C01842=1151.994,50.218,-50.534,-179.726,6.301,149.061
C01843=1151.990,50.468,-50.550,-179.724,6.302,149.061
C01844=1151.985,50.717,-50.567,-179.722,6.303,149.060
C01845=1151.979,50.966,-50.582,-179.718,6.304,149.060
C01846=1151.975,51.216,-50.597,-179.716,6.305,149.059
C01847=1151.970,51.465,-50.613,-179.713,6.307,149.059
C01848=1151.964,51.715,-50.629,-179.711,6.307,149.058
C01849=1151.960,51.965,-50.645,-179.708,6.309,149.058
C01850=1151.955,52.214,-50.661,-179.705,6.309,149.057
C01851=1151.950,52.463,-50.676,-179.703,6.310,149.057
C01852=1151.945,52.713,-50.692,-179.700,6.312,149.056
C01853=1151.940,52.962,-50.707,-179.698,6.312,149.056
C01854=1151.934,53.212,-50.723,-179.695,6.314,149.055
C01855=1151.929,53.481,-50.740,-179.692,6.315,149.054
C01856=1151.924,53.749,-50.757,-179.689,6.316,149.054
C01857=1151.918,54.018,-50.774,-179.686,6.318,149.053
C01858=1151.913,54.286,-50.791,-179.683,6.319,149.053
C01859=1151.908,54.535,-50.808,-179.681,6.320,149.052
C01860=1151.904,54.785,-50.823,-179.678,6.321,149.052
C01861=1151.898,55.034,-50.839,-179.676,6.322,149.051
C01862=1151.894,55.284,-50.855,-179.673,6.323,149.051
C01863=1151.888,55.533,-50.871,-179.670,6.324,149.050
C01864=1151.883,55.783,-50.887,-179.668,6.326,149.050
C01865=1151.878,56.032,-50.903,-179.665,6.326,149.049
C01866=1151.873,56.282,-50.919,-179.662,6.328,149.048
C01867=1151.868,56.532,-50.935,-179.660,6.329,149.048
C01868=1151.863,56.780,-50.951,-179.657,6.330,149.047
C01869=1151.858,57.030,-50.967,-179.655,6.331,149.047
C01870=1151.853,57.280,-50.983,-179.651,6.332,149.046
C01871=1151.848,57.529,-50.999,-179.649,6.333,149.046
C01872=1151.843,57.779,-51.015,-179.646,6.335,149.045
C01873=1151.838,58.028,-51.031,-179.644,6.335,149.045
C01874=1151.833,58.277,-51.047,-179.641,6.337,149.044
C01875=1151.828,58.526,-51.063,-179.638,6.337,149.044
C01876=1151.823,58.776,-51.079,-179.636,6.339,149.043
C01877=1151.818,59.025,-51.096,-179.634,6.340,149.043
C01878=1151.813,59.275,-51.111,-179.630,6.341,149.042
C01879=1151.808,59.525,-51.127,-179.628,6.342,149.042
C01880=1151.803,59.774,-51.144,-179.625,6.344,149.041
C01881=1151.798,60.024,-51.159,-179.623,6.344,149.041
C01882=1151.793,60.273,-51.176,-179.620,6.346,149.040
C01883=1151.788,60.523,-51.192,-179.617,6.346,149.039
C01884=1151.783,60.771,-51.208,-179.615,6.348,149.039
C01885=1151.779,61.021,-51.225,-179.613,6.349,149.039
C01886=1151.773,61.270,-51.240,-179.609,6.350,149.038
C01887=1151.769,61.520,-51.257,-179.607,6.351,149.037
C01888=1151.764,61.769,-51.273,-179.604,6.352,149.037
C01889=1151.759,62.019,-51.289,-179.602,6.353,149.036
C01890=1151.754,62.268,-51.305,-179.599,6.355,149.036
C01891=1151.749,62.518,-51.322,-179.596,6.356,149.035
C01892=1151.743,62.767,-51.338,-179.594,6.357,149.035
C01893=1151.739,63.017,-51.354,-179.591,6.358,149.034
C01894=1151.734,63.266,-51.371,-179.588,6.359,149.034
C01895=1151.729,63.516,-51.387,-179.585,6.361,149.033
C01896=1151.724,63.764,-51.403,-179.583,6.361,149.033
C01897=1151.719,64.014,-51.420,-179.580,6.363,149.032
C01898=1151.714,64.263,-51.435,-179.578,6.364,149.032
C01899=1151.709,64.513,-51.452,-179.575,6.365,149.031
C01900=1151.704,64.762,-51.469,-179.573,6.366,149.031
C01901=1151.699,65.012,-51.485,-179.570,6.367,149.030
C01902=1151.694,65.261,-51.501,-179.567,6.369,149.030
C01903=1151.689,65.510,-51.518,-179.564,6.370,149.029
C01904=1151.685,65.760,-51.534,-179.562,6.371,149.029
C01905=1151.679,66.009,-51.551,-179.559,6.372,149.028
C01906=1151.674,66.259,-51.567,-179.556,6.373,149.028
C01907=1151.669,66.508,-51.583,-179.554,6.374,149.027
C01908=1151.665,66.757,-51.600,-179.551,6.376,149.027
C01909=1151.660,67.007,-51.616,-179.548,6.377,149.026
C01910=1151.654,67.256,-51.633,-179.546,6.378,149.025
C01911=1151.649,67.506,-51.650,-179.543,6.379,149.025
C01912=1151.644,67.755,-51.666,-179.541,6.380,149.025
C01913=1151.640,68.004,-51.683,-179.537,6.382,149.024
C01914=1151.634,68.255,-51.699,-179.535,6.382,149.023
C01915=1151.629,68.503,-51.715,-179.533,6.384,149.023
C01916=1151.625,68.753,-51.732,-179.529,6.385,149.022
C01917=1151.620,69.002,-51.748,-179.527,6.386,149.022
C01918=1151.615,69.251,-51.766,-179.524,6.388,149.022
C01919=1151.610,69.501,-51.782,-179.522,6.388,149.021
C01920=1151.605,69.750,-51.799,-179.519,6.390,149.020
C01921=1151.599,70.000,-51.815,-179.516,6.392,149.020
C01922=1151.595,70.250,-51.832,-179.514,6.392,149.019
C01923=1151.590,70.498,-51.848,-179.511,6.394,149.019
C01924=1151.585,70.748,-51.865,-179.509,6.395,149.018
C01925=1151.580,70.998,-51.882,-179.506,6.396,149.018
C01926=1151.575,71.246,-51.898,-179.503,6.398,149.017
C01927=1151.570,71.496,-51.916,-179.501,6.399,149.017
C01928=1151.565,71.746,-51.932,-179.497,6.400,149.016
C01929=1151.560,71.994,-51.949,-179.495,6.401,149.016
C01930=1151.555,72.244,-51.966,-179.493,6.402,149.015
C01931=1151.551,72.494,-51.983,-179.489,6.404,149.015
C01932=1151.546,72.743,-51.999,-179.487,6.405,149.014
C01933=1151.540,72.992,-52.016,-179.484,6.406,149.014
C01934=1151.536,73.242,-52.033,-179.482,6.407,149.013
C01935=1151.530,73.491,-52.050,-179.479,6.408,149.013
C01936=1151.526,73.740,-52.066,-179.476,6.410,149.012
C01937=1151.521,73.990,-52.083,-179.474,6.411,149.012
C01938=1151.516,74.240,-52.100,-179.471,6.412,149.011
C01939=1151.511,74.488,-52.117,-179.468,6.413,149.011
C01940=1151.506,74.738,-52.134,-179.466,6.414,149.010
C01941=1151.501,74.988,-52.151,-179.463,6.416,149.010
C01942=1151.496,75.238,-52.168,-179.461,6.417,149.009
C01943=1151.491,75.486,-52.185,-179.458,6.418,149.009
C01944=1151.487,75.735,-52.202,-179.455,6.420,149.008
C01945=1151.481,75.985,-52.219,-179.453,6.421,149.008
C01946=1151.477,76.234,-52.235,-179.449,6.422,149.007
C01947=1151.471,76.484,-52.252,-179.447,6.424,149.007
C01948=1151.467,76.733,-52.269,-179.445,6.425,149.006
C01949=1151.461,76.983,-52.286,-179.441,6.426,149.006
C01950=1151.457,77.232,-52.304,-179.439,6.427,149.005
C01951=1151.451,77.481,-52.321,-179.436,6.428,149.005
C01952=1151.447,77.730,-52.337,-179.433,6.430,149.004
C01953=1151.442,77.980,-52.355,-179.431,6.431,149.004
C01954=1151.436,78.230,-52.372,-179.428,6.432,149.003
C01955=1151.432,78.479,-52.389,-179.425,6.434,149.003
C01956=1151.426,78.728,-52.406,-179.423,6.435,149.002
C01957=1151.422,78.977,-52.423,-179.420,6.436,149.002
C01958=1151.417,79.227,-52.440,-179.417,6.437,149.001
C01959=1151.412,79.495,-52.459,-179.414,6.439,149.001
C01960=1151.406,79.763,-52.477,-179.412,6.440,149.000
C01961=1151.401,80.032,-52.496,-179.409,6.441,149.000
C01962=1151.396,80.300,-52.514,-179.406,6.443,148.999
C01963=1151.391,80.550,-52.531,-179.403,6.444,148.999
C01964=1151.386,80.799,-52.549,-179.401,6.445,148.998
C01965=1151.381,81.048,-52.566,-179.398,6.447,148.998
C01966=1151.376,81.298,-52.583,-179.395,6.448,148.997
C01967=1151.372,81.547,-52.600,-179.393,6.449,148.997
C01968=1151.367,81.797,-52.617,-179.390,6.451,148.996
C01969=1151.361,82.045,-52.635,-179.387,6.452,148.996
C01970=1151.357,82.295,-52.652,-179.384,6.454,148.995
C01971=1151.351,82.545,-52.669,-179.382,6.455,148.995
C01972=1151.346,82.794,-52.687,-179.379,6.456,148.994
C01973=1151.342,83.043,-52.704,-179.376,6.458,148.994
C01974=1151.337,83.292,-52.722,-179.374,6.458,148.993
C01975=1151.332,83.542,-52.739,-179.371,6.460,148.993
C01976=1151.327,83.792,-52.756,-179.368,6.461,148.992
C01977=1151.322,84.041,-52.774,-179.366,6.462,148.992
C01978=1151.317,84.290,-52.790,-179.363,6.464,148.991
C01979=1151.312,84.539,-52.808,-179.360,6.465,148.991
C01980=1151.307,84.789,-52.825,-179.358,6.466,148.990
C01981=1151.302,85.038,-52.843,-179.355,6.468,148.990
C01982=1151.297,85.288,-52.860,-179.352,6.470,148.989
C01983=1151.293,85.536,-52.878,-179.349,6.471,148.989
C01984=1151.288,85.786,-52.895,-179.347,6.472,148.988
C01985=1151.283,86.035,-52.913,-179.344,6.473,148.988
C01986=1151.278,86.285,-52.930,-179.341,6.475,148.987
C01987=1151.273,86.534,-52.948,-179.339,6.476,148.987
C01988=1151.268,86.783,-52.966,-179.336,6.477,148.986
C01989=1151.263,87.033,-52.983,-179.333,6.479,148.986
C01990=1151.258,87.282,-53.001,-179.331,6.479,148.985
C01991=1151.253,87.532,-53.018,-179.328,6.481,148.985
C01992=1151.249,87.781,-53.035,-179.325,6.483,148.984
C01993=1151.244,88.030,-53.053,-179.322,6.484,148.984
C01994=1151.239,88.280,-53.071,-179.320,6.485,148.983
C01995=1151.233,88.528,-53.088,-179.317,6.487,148.983
C01996=1151.228,88.778,-53.106,-179.314,6.488,148.983
C01997=1151.224,89.027,-53.123,-179.311,6.490,148.982
C01998=1151.219,89.276,-53.141,-179.309,6.491,148.981
C01999=1151.214,89.525,-53.159,-179.306,6.492,148.981
C02000=1151.209,89.775,-53.176,-179.303,6.494,148.981
C02001=1151.204,90.024,-53.194,-179.301,6.494,148.980
C02002=1151.200,90.274,-53.213,-179.298,6.496,148.980
C02003=1151.194,90.524,-53.230,-179.295,6.498,148.979
C02004=1151.190,90.773,-53.248,-179.293,6.499,148.979
C02005=1151.185,91.022,-53.265,-179.290,6.500,148.978
C02006=1151.180,91.271,-53.283,-179.287,6.502,148.978
C02007=1151.175,91.521,-53.300,-179.284,6.503,148.977
C02008=1151.170,91.770,-53.318,-179.282,6.505,148.977
C02009=1151.165,92.019,-53.336,-179.279,6.506,148.976
C02010=1151.160,92.269,-53.354,-179.276,6.507,148.976
C02011=1151.156,92.518,-53.372,-179.274,6.509,148.975
C02012=1151.150,92.768,-53.390,-179.271,6.511,148.975
C02013=1151.145,93.017,-53.408,-179.268,6.511,148.974
C02014=1151.141,93.266,-53.426,-179.266,6.513,148.974
C02015=1151.136,93.515,-53.443,-179.263,6.514,148.973
C02016=1151.131,93.764,-53.461,-179.260,6.516,148.973
C02017=1151.126,94.013,-53.479,-179.257,6.517,148.972
C02018=1151.121,94.263,-53.497,-179.255,6.518,148.972
C02019=1151.116,94.513,-53.515,-179.252,6.520,148.972
C02020=1151.111,94.762,-53.533,-179.249,6.522,148.971
C02021=1151.106,95.011,-53.551,-179.246,6.523,148.970
C02022=1151.102,95.261,-53.569,-179.244,6.524,148.970
C02023=1151.097,95.510,-53.587,-179.241,6.526,148.970
C02024=1151.092,95.759,-53.605,-179.238,6.527,148.969
C02025=1151.087,96.008,-53.623,-179.235,6.529,148.969
C02026=1151.082,96.257,-53.641,-179.233,6.529,148.968
C02027=1151.077,96.506,-53.659,-179.230,6.531,148.968
C02028=1151.073,96.756,-53.677,-179.228,6.533,148.967
C02029=1151.068,97.006,-53.695,-179.224,6.534,148.967
C02030=1151.063,97.255,-53.713,-179.222,6.536,148.966
C02031=1151.058,97.504,-53.731,-179.220,6.537,148.966
C02032=1151.053,97.753,-53.749,-179.217,6.538,148.965
C02033=1151.048,98.002,-53.767,-179.214,6.540,148.965
C02034=1151.043,98.251,-53.785,-179.211,6.541,148.964
C02035=1151.038,98.502,-53.804,-179.208,6.543,148.964
C02036=1151.033,98.751,-53.822,-179.206,6.544,148.964
C02037=1151.028,99.000,-53.840,-179.203,6.546,148.963
C02038=1151.023,99.249,-53.858,-179.200,6.547,148.962
C02039=1151.019,99.498,-53.876,-179.197,6.549,148.962
C02040=1151.014,99.748,-53.895,-179.195,6.550,148.962
C02041=1151.010,99.997,-53.913,-179.192,6.551,148.961
C02042=1151.004,100.246,-53.932,-179.190,6.553,148.961
C02043=1150.999,100.495,-53.950,-179.187,6.554,148.960
C02044=1150.994,100.745,-53.968,-179.184,6.556,148.960
C02045=1150.990,100.994,-53.986,-179.181,6.558,148.959
C02046=1150.985,101.244,-54.004,-179.179,6.559,148.959
C02047=1150.980,101.492,-54.023,-179.176,6.560,148.959
C02048=1150.975,101.742,-54.041,-179.173,6.562,148.958
C02049=1150.970,101.992,-54.060,-179.170,6.563,148.957
C02050=1150.965,102.241,-54.077,-179.168,6.565,148.957
C02051=1150.960,102.490,-54.095,-179.165,6.567,148.957
C02052=1150.955,102.739,-54.115,-179.162,6.567,148.956
C02053=1150.951,102.989,-54.133,-179.159,6.569,148.956
C02054=1150.946,103.238,-54.151,-179.157,6.571,148.955
C02055=1150.941,103.487,-54.169,-179.154,6.572,148.955
C02056=1150.936,103.736,-54.188,-179.151,6.574,148.954
C02057=1150.931,103.986,-54.207,-179.149,6.576,148.954
C02058=1150.926,104.235,-54.225,-179.146,6.576,148.953
C02059=1150.922,104.483,-54.243,-179.143,6.578,148.953
C02060=1150.916,104.733,-54.262,-179.140,6.580,148.952
C02061=1150.912,104.983,-54.280,-179.138,6.581,148.952
C02062=1150.907,105.231,-54.299,-179.135,6.583,148.952
C02063=1150.901,105.500,-54.319,-179.132,6.584,148.951
C02064=1150.896,105.768,-54.338,-179.129,6.586,148.951
C02065=1150.891,106.037,-54.359,-179.126,6.587,148.950
C02066=1150.886,106.305,-54.379,-179.123,6.589,148.950
C02067=1150.881,106.555,-54.397,-179.120,6.591,148.949
C02068=1150.877,106.804,-54.417,-179.118,6.592,148.949
C02069=1150.872,107.053,-54.435,-179.115,6.594,148.948
C02070=1150.866,107.303,-54.453,-179.112,6.595,148.948
C02071=1150.862,107.552,-54.472,-179.110,6.596,148.947
C02072=1150.857,107.801,-54.490,-179.107,6.598,148.947
C02073=1150.852,108.050,-54.509,-179.104,6.600,148.946
C02074=1150.848,108.300,-54.528,-179.101,6.601,148.946
C02075=1150.842,108.549,-54.547,-179.099,6.603,148.946
C02076=1150.837,108.798,-54.565,-179.096,6.604,148.945
C02077=1150.833,109.047,-54.584,-179.093,6.606,148.945
C02078=1150.828,109.296,-54.603,-179.091,6.607,148.944
C02079=1150.823,109.545,-54.621,-179.088,6.609,148.944
C02080=1150.818,109.795,-54.640,-179.085,6.610,148.943
C02081=1150.813,110.044,-54.659,-179.083,6.612,148.943
C02082=1150.808,110.294,-54.678,-179.079,6.613,148.942
C02083=1150.804,110.543,-54.697,-179.077,6.615,148.942
C02084=1150.798,110.791,-54.716,-179.074,6.617,148.942
C02085=1150.794,111.041,-54.734,-179.071,6.618,148.941
C02086=1150.789,111.290,-54.754,-179.069,6.619,148.941
C02087=1150.784,111.540,-54.772,-179.066,6.621,148.940
C02088=1150.779,111.789,-54.791,-179.063,6.622,148.940
C02089=1150.775,112.037,-54.810,-179.060,6.624,148.939
C02090=1150.769,112.288,-54.829,-179.058,6.626,148.939
C02091=1150.765,112.536,-54.848,-179.055,6.627,148.938
C02092=1150.760,112.786,-54.867,-179.052,6.629,148.938
C02093=1150.755,113.035,-54.885,-179.049,6.631,148.938
C02094=1150.750,113.285,-54.905,-179.047,6.633,148.937
C02095=1150.746,113.533,-54.924,-179.044,6.634,148.937
C02096=1150.741,113.783,-54.942,-179.041,6.635,148.936
C02097=1150.736,114.032,-54.961,-179.039,6.636,148.936
C02098=1150.731,114.281,-54.981,-179.036,6.638,148.935
C02099=1150.726,114.530,-55.000,-179.033,6.640,148.935
C02100=1150.721,114.779,-55.018,-179.031,6.642,148.935
C02101=1150.716,115.029,-55.038,-179.028,6.643,148.934
C02102=1150.712,115.278,-55.056,-179.025,6.645,148.934
C02103=1150.707,115.527,-55.076,-179.022,6.646,148.933
C02104=1150.701,115.777,-55.095,-179.019,6.648,148.933
C02105=1150.697,116.026,-55.114,-179.016,6.650,148.932
C02106=1150.692,116.275,-55.133,-179.014,6.651,148.932
C02107=1150.688,116.524,-55.152,-179.011,6.653,148.931
C02108=1150.683,116.773,-55.171,-179.008,6.655,148.931
C02109=1150.678,117.022,-55.191,-179.006,6.656,148.931
C02110=1150.673,117.272,-55.209,-179.003,6.657,148.930
C02111=1150.668,117.521,-55.229,-179.000,6.659,148.930
C02112=1150.664,117.771,-55.248,-178.997,6.660,148.929
C02113=1150.659,118.019,-55.267,-178.995,6.662,148.929
C02114=1150.654,118.269,-55.287,-178.992,6.664,148.928
C02115=1150.649,118.518,-55.306,-178.989,6.666,148.928
C02116=1150.644,118.767,-55.326,-178.987,6.667,148.928
C02117=1150.640,119.016,-55.344,-178.984,6.669,148.927
C02118=1150.635,119.265,-55.364,-178.981,6.671,148.927
C02119=1150.629,119.514,-55.383,-178.978,6.672,148.926
C02120=1150.625,119.764,-55.402,-178.975,6.674,148.926
C02121=1150.621,120.013,-55.422,-178.973,6.675,148.925
C02122=1150.615,120.262,-55.441,-178.970,6.677,148.925
C02123=1150.611,120.512,-55.461,-178.967,6.679,148.925
C02124=1150.605,120.760,-55.480,-178.964,6.681,148.924
C02125=1150.601,121.010,-55.499,-178.962,6.682,148.924
C02126=1150.597,121.259,-55.519,-178.959,6.684,148.923
C02127=1150.591,121.508,-55.538,-178.956,6.686,148.923
C02128=1150.586,121.758,-55.558,-178.953,6.687,148.923
C02129=1150.582,122.006,-55.577,-178.950,6.689,148.922
C02130=1150.577,122.256,-55.596,-178.948,6.690,148.922
C02131=1150.572,122.505,-55.616,-178.945,6.691,148.921
C02132=1150.567,122.754,-55.635,-178.943,6.693,148.921
C02133=1150.562,123.004,-55.655,-178.940,6.695,148.920
C02134=1150.558,123.253,-55.674,-178.937,6.696,148.920
C02135=1150.553,123.501,-55.694,-178.935,6.698,148.920
C02136=1150.549,123.751,-55.714,-178.932,6.700,148.919
C02137=1150.544,124.000,-55.733,-178.929,6.701,148.919
C02138=1150.538,124.249,-55.753,-178.926,6.703,148.918
C02139=1150.534,124.499,-55.772,-178.924,6.705,148.918
C02140=1150.529,124.748,-55.792,-178.921,6.707,148.918
C02141=1150.524,124.997,-55.812,-178.918,6.708,148.917
C02142=1150.519,125.246,-55.831,-178.915,6.710,148.917
C02143=1150.515,125.496,-55.851,-178.912,6.711,148.916
C02144=1150.510,125.744,-55.870,-178.910,6.713,148.916
C02145=1150.505,125.993,-55.890,-178.907,6.715,148.915
C02146=1150.501,126.243,-55.910,-178.904,6.716,148.915
C02147=1150.495,126.492,-55.929,-178.901,6.718,148.915
C02148=1150.491,126.741,-55.949,-178.899,6.720,148.914
C02149=1150.486,126.990,-55.969,-178.896,6.722,148.914
C02150=1150.481,127.240,-55.989,-178.893,6.723,148.913
C02151=1150.476,127.489,-56.008,-178.891,6.725,148.913
C02152=1150.472,127.738,-56.028,-178.888,6.727,148.913
C02153=1150.467,127.987,-56.048,-178.885,6.728,148.912
C02154=1150.462,128.237,-56.068,-178.882,6.730,148.912
C02155=1150.457,128.485,-56.088,-178.880,6.732,148.911
C02156=1150.452,128.735,-56.107,-178.877,6.734,148.911
C02157=1150.448,128.984,-56.127,-178.874,6.735,148.911
C02158=1150.443,129.233,-56.148,-178.871,6.737,148.910
C02159=1150.438,129.482,-56.167,-178.868,6.738,148.910
C02160=1150.433,129.731,-56.187,-178.865,6.741,148.909
C02161=1150.429,129.981,-56.207,-178.862,6.743,148.909
C02162=1150.424,130.230,-56.226,-178.860,6.744,148.908
C02163=1150.419,130.478,-56.246,-178.857,6.746,148.908
C02164=1150.414,130.728,-56.266,-178.854,6.748,148.908
C02165=1150.410,130.977,-56.287,-178.851,6.749,148.907
C02166=1150.405,131.226,-56.306,-178.849,6.751,148.907
C02167=1150.400,131.495,-56.329,-178.846,6.753,148.906
C02168=1150.395,131.763,-56.350,-178.843,6.755,148.906
C02169=1150.389,132.032,-56.371,-178.840,6.757,148.906
C02170=1150.384,132.300,-56.393,-178.837,6.758,148.905
C02171=1150.380,132.550,-56.413,-178.834,6.760,148.905
C02172=1150.375,132.798,-56.433,-178.831,6.762,148.904
C02173=1150.369,133.048,-56.453,-178.829,6.764,148.904
C02174=1150.365,133.297,-56.473,-178.826,6.765,148.903
C02175=1150.360,133.547,-56.493,-178.823,6.767,148.903
C02176=1150.355,133.796,-56.513,-178.821,6.769,148.903
C02177=1150.351,134.045,-56.534,-178.818,6.770,148.902
C02178=1150.346,134.293,-56.553,-178.815,6.772,148.902
C02179=1150.341,134.543,-56.574,-178.812,6.774,148.901
C02180=1150.336,134.792,-56.594,-178.810,6.776,148.901
C02181=1150.331,135.041,-56.614,-178.806,6.778,148.901
C02182=1150.327,135.290,-56.634,-178.804,6.780,148.900
C02183=1150.322,135.539,-56.655,-178.801,6.781,148.900
C02184=1150.317,135.789,-56.675,-178.798,6.783,148.900
C02185=1150.313,136.038,-56.695,-178.796,6.785,148.899
C02186=1150.308,136.286,-56.715,-178.793,6.787,148.899
C02187=1150.303,136.536,-56.735,-178.790,6.788,148.898
C02188=1150.298,136.785,-56.756,-178.787,6.790,148.898
C02189=1150.293,137.034,-56.776,-178.785,6.792,148.898
C02190=1150.289,137.283,-56.797,-178.782,6.793,148.897
C02191=1150.284,137.532,-56.816,-178.779,6.795,148.897
C02192=1150.279,137.782,-56.837,-178.777,6.797,148.896
C02193=1150.274,138.031,-56.858,-178.774,6.799,148.896
C02194=1150.270,138.280,-56.878,-178.771,6.801,148.896
C02195=1150.266,138.529,-56.899,-178.768,6.803,148.895
C02196=1150.260,138.778,-56.919,-178.765,6.805,148.895
C02197=1150.256,139.027,-56.939,-178.762,6.806,148.894
C02198=1150.251,139.276,-56.960,-178.760,6.808,148.894
C02199=1150.246,139.526,-56.981,-178.757,6.810,148.894
C02200=1150.242,139.775,-57.001,-178.754,6.811,148.893
C02201=1150.237,140.023,-57.021,-178.752,6.813,148.893
C02202=1150.232,140.273,-57.042,-178.749,6.815,148.893
C02203=1150.227,140.522,-57.062,-178.746,6.817,148.892
C02204=1150.222,140.772,-57.083,-178.743,6.819,148.892
C02205=1150.218,141.021,-57.103,-178.740,6.821,148.891
C02206=1150.213,141.269,-57.124,-178.738,6.823,148.891
C02207=1150.208,141.519,-57.145,-178.735,6.825,148.891
C02208=1150.204,141.768,-57.165,-178.732,6.826,148.890
C02209=1150.198,142.017,-57.186,-178.730,6.828,148.890
C02210=1150.194,142.266,-57.206,-178.727,6.830,148.890
C02211=1150.189,142.515,-57.227,-178.724,6.831,148.889
C02212=1150.184,142.764,-57.248,-178.721,6.834,148.889
C02213=1150.180,143.013,-57.268,-178.718,6.836,148.889
C02214=1150.175,143.262,-57.289,-178.716,6.837,148.888
C02215=1150.170,143.511,-57.309,-178.713,6.839,148.888
C02216=1150.165,143.760,-57.330,-178.710,6.841,148.887
C02217=1150.161,144.009,-57.351,-178.707,6.843,148.887
C02218=1150.155,144.259,-57.372,-178.705,6.844,148.887
C02219=1150.151,144.508,-57.392,-178.701,6.847,148.886
C02220=1150.147,144.757,-57.412,-178.699,6.849,148.886
C02221=1150.142,145.005,-57.434,-178.696,6.850,148.885
C02222=1150.137,145.254,-57.455,-178.693,6.852,148.885
C02223=1150.132,145.503,-57.475,-178.691,6.854,148.885
C02224=1150.127,145.753,-57.496,-178.688,6.855,148.884
C02225=1150.122,146.002,-57.517,-178.685,6.857,148.884
C02226=1150.118,146.252,-57.538,-178.682,6.860,148.884
C02227=1150.113,146.501,-57.558,-178.680,6.862,148.883
C02228=1150.109,146.749,-57.580,-178.677,6.863,148.883
C02229=1150.104,146.998,-57.601,-178.674,6.865,148.883
C02230=1150.099,147.247,-57.621,-178.672,6.867,148.882
C02231=1150.095,147.496,-57.642,-178.669,6.869,148.882
C02232=1150.090,147.745,-57.664,-178.666,6.871,148.881
C02233=1150.085,147.994,-57.685,-178.663,6.873,148.881
C02234=1150.081,148.244,-57.705,-178.660,6.875,148.881
C02235=1150.076,148.493,-57.726,-178.657,6.876,148.880
C02236=1150.071,148.742,-57.748,-178.655,6.878,148.880
C02237=1150.066,148.991,-57.768,-178.652,6.880,148.880
C02238=1150.061,149.240,-57.789,-178.649,6.883,148.879
C02239=1150.057,149.489,-57.810,-178.647,6.884,148.879
C02240=1150.052,149.738,-57.831,-178.644,6.886,148.879
C02241=1150.047,149.988,-57.853,-178.641,6.888,148.878
C02242=1150.043,150.237,-57.873,-178.638,6.890,148.878
C02243=1150.038,150.485,-57.895,-178.636,6.891,148.877
C02244=1150.033,150.734,-57.916,-178.632,6.894,148.877
C02245=1150.028,150.983,-57.937,-178.630,6.896,148.877
C02246=1150.023,151.232,-57.958,-178.627,6.897,148.876
C02247=1150.019,151.482,-57.979,-178.624,6.899,148.876
C02248=1150.014,151.731,-58.001,-178.622,6.901,148.876
C02249=1150.009,151.980,-58.021,-178.619,6.904,148.875
C02250=1150.005,152.228,-58.043,-178.616,6.905,148.875
C02251=1150.000,152.478,-58.064,-178.613,6.907,148.875
C02252=1149.995,152.727,-58.086,-178.611,6.909,148.874
C02253=1149.991,152.976,-58.106,-178.608,6.910,148.874
C02254=1149.986,153.225,-58.127,-178.605,6.913,148.874
C02255=1149.981,153.474,-58.149,-178.602,6.915,148.873
C02256=1149.976,153.724,-58.170,-178.599,6.916,148.873
C02257=1149.971,153.972,-58.192,-178.597,6.919,148.873
C02258=1149.967,154.221,-58.213,-178.594,6.920,148.872
C02259=1149.962,154.470,-58.234,-178.591,6.923,148.872
C02260=1149.958,154.719,-58.256,-178.588,6.925,148.872
C02261=1149.952,154.968,-58.277,-178.586,6.926,148.871
C02262=1149.948,155.217,-58.299,-178.583,6.928,148.871
C02263=1149.944,155.467,-58.319,-178.580,6.930,148.870
C02264=1149.939,155.715,-58.341,-178.577,6.933,148.870
C02265=1149.934,155.964,-58.363,-178.575,6.934,148.870
C02266=1149.929,156.213,-58.384,-178.572,6.936,148.869
C02267=1149.925,156.463,-58.406,-178.569,6.938,148.869
C02268=1149.920,156.711,-58.427,-178.566,6.940,148.869
C02269=1149.915,156.961,-58.448,-178.563,6.942,148.868
C02270=1149.911,157.210,-58.470,-178.561,6.944,148.868
C02271=1149.906,157.479,-58.493,-178.557,6.946,148.868
C02272=1149.900,157.747,-58.516,-178.555,6.948,148.867
C02273=1149.895,158.016,-58.540,-178.551,6.951,148.867
C02274=1149.890,158.285,-58.563,-178.549,6.952,148.866
C02275=1149.886,158.534,-58.584,-178.546,6.954,148.866
C02276=1149.881,158.783,-58.606,-178.543,6.957,148.866
C02277=1149.876,159.032,-58.627,-178.540,6.959,148.866
C02278=1149.872,159.282,-58.649,-178.538,6.960,148.865
C02279=1149.867,159.530,-58.671,-178.535,6.962,148.865
C02280=1149.863,159.780,-58.693,-178.532,6.965,148.864
C02281=1149.857,160.029,-58.714,-178.529,6.967,148.864
C02282=1149.853,160.277,-58.736,-178.527,6.968,148.864
C02283=1149.848,160.527,-58.758,-178.524,6.970,148.864
C02284=1149.843,160.775,-58.779,-178.521,6.973,148.863
C02285=1149.839,161.024,-58.801,-178.518,6.974,148.863
C02286=1149.834,161.273,-58.823,-178.515,6.976,148.862
C02287=1149.829,161.522,-58.845,-178.513,6.979,148.862
C02288=1149.825,161.772,-58.866,-178.510,6.981,148.862
C02289=1149.820,162.021,-58.888,-178.507,6.983,148.862
C02290=1149.816,162.270,-58.910,-178.504,6.984,148.861
C02291=1149.811,162.519,-58.931,-178.501,6.987,148.861
C02292=1149.806,162.767,-58.953,-178.499,6.989,148.861
C02293=1149.802,163.017,-58.975,-178.496,6.991,148.860
C02294=1149.796,163.266,-58.997,-178.493,6.993,148.860
C02295=1149.792,163.515,-59.019,-178.490,6.995,148.860
C02296=1149.787,163.764,-59.041,-178.488,6.997,148.859
C02297=1149.783,164.013,-59.063,-178.485,6.999,148.859
C02298=1149.778,164.262,-59.085,-178.482,7.001,148.859
C02299=1149.774,164.511,-59.107,-178.479,7.003,148.858
C02300=1149.769,164.760,-59.129,-178.477,7.005,148.858
C02301=1149.764,165.009,-59.151,-178.473,7.007,148.858
C02302=1149.760,165.258,-59.172,-178.471,7.009,148.857
C02303=1149.754,165.506,-59.195,-178.468,7.011,148.857
C02304=1149.750,165.756,-59.217,-178.466,7.013,148.857
C02305=1149.745,166.004,-59.238,-178.462,7.015,148.856
C02306=1149.740,166.254,-59.260,-178.460,7.017,148.856
C02307=1149.736,166.502,-59.283,-178.457,7.019,148.856
C02308=1149.732,166.751,-59.305,-178.454,7.022,148.855
C02309=1149.726,167.000,-59.327,-178.451,7.023,148.855
C02310=1149.722,167.249,-59.349,-178.449,7.025,148.855
C02311=1149.718,167.499,-59.371,-178.446,7.028,148.855
C02312=1149.713,167.747,-59.393,-178.443,7.030,148.854
C02313=1149.708,167.997,-59.416,-178.441,7.032,148.854
C02314=1149.703,168.245,-59.438,-178.437,7.034,148.854
C02315=1149.699,168.494,-59.460,-178.435,7.036,148.853
C02316=1149.694,168.743,-59.482,-178.432,7.038,148.853
C02317=1149.689,168.993,-59.504,-178.429,7.040,148.853
C02318=1149.684,169.241,-59.527,-178.426,7.042,148.852
C02319=1149.680,169.490,-59.549,-178.424,7.044,148.852
C02320=1149.675,169.739,-59.570,-178.421,7.047,148.852
C02321=1149.670,169.988,-59.593,-178.418,7.049,148.851
C02322=1149.666,170.237,-59.616,-178.415,7.050,148.851
C02323=1149.661,170.486,-59.638,-178.413,7.053,148.851
C02324=1149.656,170.735,-59.660,-178.410,7.055,148.851
C02325=1149.652,170.983,-59.683,-178.407,7.057,148.850
C02326=1149.648,171.233,-59.705,-178.404,7.059,148.850
C02327=1149.643,171.482,-59.727,-178.402,7.061,148.850
C02328=1149.638,171.730,-59.750,-178.399,7.063,148.849
C02329=1149.634,171.980,-59.772,-178.396,7.066,148.849
C02330=1149.628,172.229,-59.794,-178.393,7.067,148.849
C02331=1149.624,172.477,-59.817,-178.391,7.069,148.848
C02332=1149.619,172.727,-59.839,-178.388,7.072,148.848
C02333=1149.615,172.975,-59.862,-178.385,7.074,148.848
C02334=1149.610,173.224,-59.884,-178.383,7.076,148.848
C02335=1149.606,173.474,-59.907,-178.379,7.078,148.847
C02336=1149.601,173.722,-59.929,-178.377,7.080,148.847
C02337=1149.596,173.972,-59.952,-178.373,7.083,148.846
C02338=1149.592,174.221,-59.974,-178.371,7.085,148.846
C02339=1149.586,174.469,-59.997,-178.369,7.086,148.846
C02340=1149.582,174.718,-60.019,-178.365,7.089,148.846
C02341=1149.578,174.968,-60.041,-178.363,7.091,148.845
C02342=1149.573,175.216,-60.064,-178.360,7.093,148.845
C02343=1149.569,175.465,-60.087,-178.357,7.095,148.845
C02344=1149.564,175.714,-60.110,-178.354,7.097,148.844
C02345=1149.559,175.962,-60.132,-178.352,7.100,148.844
C02346=1149.554,176.212,-60.155,-178.349,7.102,148.844
C02347=1149.550,176.461,-60.178,-178.346,7.103,148.844
C02348=1149.545,176.710,-60.200,-178.343,7.106,148.843
C02349=1149.541,176.958,-60.223,-178.341,7.108,148.843
C02350=1149.536,177.207,-60.246,-178.338,7.110,148.843
C02351=1149.532,177.457,-60.268,-178.335,7.113,148.843
C02352=1149.526,177.705,-60.291,-178.332,7.114,148.842
C02353=1149.522,177.954,-60.314,-178.329,7.117,148.842
C02354=1149.517,178.203,-60.336,-178.327,7.119,148.842
C02355=1149.513,178.452,-60.360,-178.324,7.121,148.841
C02356=1149.508,178.700,-60.382,-178.321,7.123,148.841
C02357=1149.503,178.950,-60.405,-178.319,7.125,148.841
C02358=1149.499,179.199,-60.428,-178.315,7.128,148.841
C02359=1149.494,179.448,-60.451,-178.313,7.130,148.840
C02360=1149.489,179.696,-60.474,-178.311,7.132,148.840
C02361=1149.485,179.946,-60.496,-178.307,7.134,148.840
C02362=1149.480,180.195,-60.519,-178.305,7.136,148.839
C02363=1149.476,180.443,-60.542,-178.302,7.139,148.839
C02364=1149.471,180.692,-60.565,-178.299,7.141,148.839
C02365=1149.466,180.941,-60.588,-178.296,7.143,148.838
C02366=1149.462,181.190,-60.611,-178.294,7.145,148.838
C02367=1149.457,181.439,-60.634,-178.291,7.147,148.838
C02368=1149.453,181.688,-60.657,-178.288,7.150,148.838
C02369=1149.449,181.937,-60.680,-178.285,7.152,148.837
C02370=1149.444,182.186,-60.703,-178.282,7.154,148.837
C02371=1149.439,182.434,-60.726,-178.279,7.156,148.837
C02372=1149.435,182.683,-60.749,-178.277,7.159,148.837
C02373=1149.430,182.933,-60.772,-178.274,7.161,148.836
C02374=1149.425,183.182,-60.795,-178.271,7.162,148.836
C02375=1149.420,183.451,-60.821,-178.268,7.165,148.836
C02376=1149.415,183.720,-60.845,-178.265,7.168,148.835
C02377=1149.410,183.990,-60.870,-178.262,7.171,148.835
C02378=1149.405,184.260,-60.895,-178.259,7.172,148.835
C02379=1149.400,184.509,-60.919,-178.256,7.175,148.835
C02380=1149.396,184.757,-60.941,-178.254,7.177,148.834
C02381=1149.391,185.006,-60.965,-178.250,7.179,148.834
C02382=1149.387,185.255,-60.988,-178.248,7.182,148.834
C02383=1149.382,185.505,-61.012,-178.245,7.184,148.833
C02384=1149.378,185.753,-61.034,-178.243,7.186,148.833
C02385=1149.373,186.002,-61.058,-178.239,7.189,148.833
C02386=1149.369,186.251,-61.081,-178.237,7.190,148.833
C02387=1149.363,186.500,-61.104,-178.235,7.193,148.833
C02388=1149.359,186.748,-61.128,-178.231,7.195,148.832
C02389=1149.354,186.997,-61.151,-178.229,7.197,148.832
C02390=1149.349,187.246,-61.175,-178.226,7.200,148.832
C02391=1149.345,187.495,-61.198,-178.223,7.202,148.831
C02392=1149.341,187.744,-61.221,-178.220,7.204,148.831
C02393=1149.336,187.993,-61.244,-178.218,7.206,148.831
C02394=1149.331,188.242,-61.268,-178.215,7.209,148.831
C02395=1149.327,188.490,-61.292,-178.212,7.211,148.830
C02396=1149.322,188.739,-61.315,-178.209,7.213,148.830
C02397=1149.318,188.988,-61.338,-178.207,7.215,148.830
C02398=1149.313,189.237,-61.362,-178.203,7.218,148.830
C02399=1149.308,189.486,-61.385,-178.201,7.220,148.829
C02400=1149.304,189.735,-61.409,-178.198,7.223,148.829
C02401=1149.299,189.984,-61.433,-178.196,7.225,148.829
C02402=1149.294,190.233,-61.456,-178.192,7.227,148.829
C02403=1149.290,190.482,-61.479,-178.190,7.229,148.828
C02404=1149.286,190.730,-61.503,-178.187,7.232,148.828
C02405=1149.281,190.979,-61.526,-178.184,7.234,148.828
C02406=1149.277,191.228,-61.550,-178.181,7.237,148.828
C02407=1149.272,191.477,-61.574,-178.179,7.238,148.827
C02408=1149.268,191.726,-61.597,-178.176,7.241,148.827
C02409=1149.263,191.975,-61.620,-178.173,7.243,148.827
C02410=1149.258,192.223,-61.645,-178.170,7.246,148.827
C02411=1149.253,192.472,-61.668,-178.168,7.248,148.826
C02412=1149.248,192.721,-61.692,-178.164,7.250,148.826
C02413=1149.244,192.970,-61.716,-178.162,7.252,148.826
C02414=1149.239,193.219,-61.739,-178.159,7.255,148.826
C02415=1149.235,193.467,-61.763,-178.157,7.257,148.825
C02416=1149.230,193.716,-61.787,-178.153,7.260,148.825
C02417=1149.226,193.965,-61.811,-178.151,7.262,148.825
C02418=1149.221,194.214,-61.834,-178.148,7.264,148.825
C02419=1149.217,194.462,-61.858,-178.146,7.266,148.825
C02420=1149.212,194.711,-61.881,-178.142,7.269,148.824
C02421=1149.208,194.960,-61.906,-178.140,7.271,148.824
C02422=1149.203,195.209,-61.929,-178.137,7.274,148.824
C02423=1149.198,195.458,-61.954,-178.135,7.276,148.824
C02424=1149.194,195.707,-61.977,-178.131,7.278,148.823
C02425=1149.189,195.956,-62.001,-178.128,7.281,148.823
C02426=1149.185,196.205,-62.025,-178.126,7.283,148.823
C02427=1149.180,196.453,-62.049,-178.123,7.285,148.822
C02428=1149.175,196.702,-62.072,-178.120,7.288,148.822
C02429=1149.171,196.951,-62.097,-178.117,7.290,148.822
C02430=1149.166,197.200,-62.121,-178.115,7.292,148.822
C02431=1149.162,197.449,-62.145,-178.112,7.295,148.822
C02432=1149.157,197.697,-62.169,-178.110,7.297,148.821
C02433=1149.153,197.946,-62.193,-178.106,7.299,148.821
C02434=1149.148,198.195,-62.217,-178.104,7.302,148.821
C02435=1149.143,198.443,-62.241,-178.101,7.304,148.821
C02436=1149.139,198.693,-62.265,-178.098,7.307,148.821
C02437=1149.135,198.942,-62.289,-178.095,7.309,148.820
C02438=1149.130,199.190,-62.313,-178.092,7.312,148.820
C02439=1149.125,199.439,-62.337,-178.090,7.313,148.820
C02440=1149.120,199.688,-62.361,-178.087,7.316,148.820
C02441=1149.117,199.937,-62.385,-178.084,7.318,148.819
C02442=1149.112,200.186,-62.410,-178.082,7.321,148.819
C02443=1149.107,200.434,-62.434,-178.079,7.323,148.819
C02444=1149.103,200.682,-62.458,-178.076,7.326,148.819
C02445=1149.098,200.931,-62.481,-178.073,7.329,148.819
C02446=1149.094,201.181,-62.506,-178.071,7.330,148.818
C02447=1149.089,201.429,-62.530,-178.068,7.333,148.818
C02448=1149.085,201.678,-62.554,-178.065,7.335,148.818
C02449=1149.080,201.926,-62.579,-178.062,7.338,148.818
C02450=1149.076,202.176,-62.604,-178.059,7.340,148.817
C02451=1149.071,202.425,-62.627,-178.057,7.343,148.817
C02452=1149.066,202.673,-62.652,-178.054,7.345,148.817
C02453=1149.062,202.922,-62.676,-178.051,7.347,148.817
C02454=1149.057,203.171,-62.701,-178.048,7.350,148.816
C02455=1149.053,203.420,-62.725,-178.046,7.352,148.816
C02456=1149.048,203.668,-62.749,-178.043,7.355,148.816
C02457=1149.044,203.917,-62.774,-178.040,7.357,148.816
C02458=1149.039,204.166,-62.798,-178.038,7.359,148.816
C02459=1149.034,204.415,-62.823,-178.034,7.362,148.815
C02460=1149.030,204.663,-62.847,-178.032,7.364,148.815
C02461=1149.026,204.912,-62.871,-178.029,7.367,148.815
C02462=1149.021,205.161,-62.896,-178.026,7.370,148.815
C02463=1149.016,205.409,-62.920,-178.023,7.371,148.815
C02464=1149.012,205.659,-62.945,-178.021,7.374,148.814
C02465=1149.008,205.907,-62.969,-178.018,7.377,148.814
C02466=1149.002,206.156,-62.994,-178.015,7.379,148.814
C02467=1148.999,206.405,-63.018,-178.012,7.382,148.814
C02468=1148.994,206.654,-63.043,-178.010,7.384,148.814
C02469=1148.989,206.902,-63.067,-178.007,7.387,148.813
C02470=1148.985,207.151,-63.092,-178.004,7.389,148.813
C02471=1148.980,207.399,-63.117,-178.001,7.391,148.813
C02472=1148.975,207.648,-63.141,-177.998,7.394,148.813
C02473=1148.971,207.897,-63.166,-177.995,7.397,148.813
C02474=1148.966,208.146,-63.190,-177.993,7.399,148.812
C02475=1148.961,208.394,-63.215,-177.990,7.402,148.812
C02476=1148.958,208.644,-63.240,-177.988,7.403,148.812
C02477=1148.953,208.892,-63.265,-177.985,7.406,148.812
C02478=1148.949,209.141,-63.289,-177.981,7.409,148.812
C02479=1148.943,209.411,-63.317,-177.979,7.412,148.811
C02480=1148.938,209.682,-63.344,-177.975,7.414,148.811
C02481=1148.933,209.952,-63.371,-177.973,7.417,148.811
C02482=1148.929,210.223,-63.398,-177.969,7.420,148.811
C02483=1148.924,210.472,-63.422,-177.967,7.422,148.811
C02484=1148.919,210.720,-63.446,-177.964,7.425,148.811
C02485=1148.915,210.969,-63.472,-177.961,7.428,148.810
C02486=1148.911,211.218,-63.496,-177.959,7.430,148.810
C02487=1148.906,211.467,-63.521,-177.956,7.432,148.810
C02488=1148.901,211.715,-63.547,-177.953,7.434,148.810
C02489=1148.897,211.964,-63.571,-177.951,7.437,148.810
C02490=1148.892,212.213,-63.596,-177.947,7.440,148.809
C02491=1148.888,212.462,-63.621,-177.945,7.442,148.809
C02492=1148.883,212.710,-63.646,-177.942,7.445,148.809
C02493=1148.879,212.958,-63.671,-177.939,7.447,148.809
C02494=1148.874,213.208,-63.696,-177.937,7.449,148.809
C02495=1148.869,213.456,-63.721,-177.934,7.452,148.808
C02496=1148.866,213.705,-63.746,-177.931,7.455,148.808
C02497=1148.861,213.954,-63.770,-177.929,7.457,148.808
C02498=1148.856,214.202,-63.796,-177.926,7.460,148.808
C02499=1148.851,214.451,-63.821,-177.923,7.463,148.808
C02500=1148.848,214.700,-63.846,-177.920,7.465,148.807
C02501=1148.843,214.948,-63.871,-177.918,7.468,148.807
C02502=1148.838,215.197,-63.896,-177.914,7.470,148.807
C02503=1148.833,215.446,-63.921,-177.911,7.473,148.807
C02504=1148.829,215.695,-63.947,-177.909,7.475,148.807
C02505=1148.826,215.943,-63.972,-177.906,7.478,148.807
C02506=1148.820,216.192,-63.997,-177.903,7.481,148.806
C02507=1148.816,216.441,-64.022,-177.901,7.483,148.806
C02508=1148.811,216.689,-64.047,-177.898,7.485,148.806
C02509=1148.807,216.938,-64.073,-177.895,7.488,148.806
C02510=1148.802,217.186,-64.098,-177.893,7.490,148.806
C02511=1148.797,217.436,-64.123,-177.889,7.493,148.805
C02512=1148.793,217.684,-64.148,-177.887,7.496,148.805
C02513=1148.789,217.932,-64.174,-177.884,7.499,148.805
C02514=1148.785,218.182,-64.199,-177.881,7.501,148.805
C02515=1148.780,218.430,-64.224,-177.878,7.503,148.805
C02516=1148.776,218.679,-64.250,-177.876,7.506,148.805
C02517=1148.770,218.927,-64.275,-177.873,7.508,148.805
C02518=1148.766,219.176,-64.300,-177.870,7.511,148.804
C02519=1148.762,219.425,-64.326,-177.867,7.514,148.804
C02520=1148.757,219.673,-64.352,-177.865,7.517,148.804
C02521=1148.753,219.923,-64.377,-177.862,7.519,148.804
C02522=1148.748,220.171,-64.402,-177.859,7.522,148.804
C02523=1148.744,220.419,-64.428,-177.856,7.524,148.804
C02524=1148.740,220.668,-64.453,-177.853,7.527,148.803
C02525=1148.735,220.916,-64.478,-177.851,7.529,148.803
C02526=1148.731,221.165,-64.503,-177.848,7.532,148.803
C02527=1148.727,221.414,-64.529,-177.845,7.535,148.803
C02528=1148.721,221.663,-64.555,-177.843,7.537,148.803
C02529=1148.717,221.912,-64.581,-177.840,7.540,148.803
C02530=1148.713,222.160,-64.607,-177.837,7.543,148.802
C02531=1148.708,222.408,-64.632,-177.834,7.546,148.802
C02532=1148.703,222.657,-64.658,-177.832,7.547,148.802
C02533=1148.699,222.906,-64.683,-177.829,7.550,148.802
C02534=1148.694,223.154,-64.709,-177.826,7.553,148.802
C02535=1148.690,223.403,-64.735,-177.823,7.556,148.802
C02536=1148.686,223.652,-64.760,-177.820,7.558,148.801
C02537=1148.682,223.901,-64.786,-177.818,7.561,148.801
C02538=1148.677,224.149,-64.811,-177.815,7.564,148.801
C02539=1148.673,224.397,-64.837,-177.812,7.567,148.801
C02540=1148.668,224.646,-64.863,-177.809,7.568,148.801
C02541=1148.664,224.894,-64.888,-177.807,7.571,148.801
C02542=1148.659,225.143,-64.915,-177.804,7.574,148.801
C02543=1148.654,225.392,-64.940,-177.801,7.577,148.801
C02544=1148.650,225.641,-64.966,-177.798,7.580,148.800
C02545=1148.645,225.889,-64.992,-177.796,7.582,148.800
C02546=1148.641,226.138,-65.017,-177.793,7.585,148.800
C02547=1148.637,226.387,-65.043,-177.790,7.588,148.800
C02548=1148.632,226.636,-65.069,-177.787,7.590,148.800
C02549=1148.627,226.884,-65.095,-177.785,7.592,148.800
C02550=1148.623,227.133,-65.121,-177.782,7.595,148.799
C02551=1148.619,227.381,-65.147,-177.779,7.598,148.799
C02552=1148.615,227.630,-65.173,-177.776,7.601,148.799
C02553=1148.610,227.879,-65.199,-177.773,7.604,148.799
C02554=1148.605,228.127,-65.224,-177.771,7.606,148.799
C02555=1148.601,228.376,-65.250,-177.768,7.609,148.799
C02556=1148.597,228.624,-65.277,-177.765,7.612,148.799
C02557=1148.592,228.873,-65.303,-177.762,7.615,148.799
C02558=1148.588,229.122,-65.329,-177.759,7.617,148.798
C02559=1148.583,229.370,-65.354,-177.757,7.619,148.798
C02560=1148.579,229.618,-65.381,-177.754,7.622,148.798
C02561=1148.574,229.867,-65.407,-177.751,7.625,148.798
C02562=1148.570,230.116,-65.433,-177.748,7.628,148.798
C02563=1148.566,230.364,-65.459,-177.745,7.631,148.798
C02564=1148.561,230.613,-65.486,-177.743,7.633,148.798
C02565=1148.556,230.862,-65.511,-177.740,7.636,148.797
C02566=1148.552,231.110,-65.537,-177.737,7.639,148.797
C02567=1148.547,231.359,-65.564,-177.735,7.641,148.797
C02568=1148.543,231.608,-65.590,-177.731,7.644,148.797
C02569=1148.539,231.856,-65.616,-177.729,7.646,148.797
C02570=1148.534,232.105,-65.642,-177.726,7.649,148.797
C02571=1148.530,232.353,-65.669,-177.724,7.652,148.797
C02572=1148.525,232.602,-65.695,-177.721,7.655,148.797
C02573=1148.521,232.851,-65.721,-177.718,7.658,148.797
C02574=1148.516,233.099,-65.747,-177.715,7.660,148.796
C02575=1148.511,233.348,-65.773,-177.713,7.663,148.796
C02576=1148.508,233.596,-65.800,-177.710,7.665,148.796
C02577=1148.503,233.845,-65.826,-177.707,7.668,148.796
C02578=1148.499,234.093,-65.853,-177.704,7.671,148.796
C02579=1148.494,234.342,-65.879,-177.701,7.674,148.796
C02580=1148.490,234.590,-65.905,-177.699,7.677,148.796
C02581=1148.486,234.839,-65.932,-177.696,7.679,148.795
C02582=1148.481,235.088,-65.958,-177.693,7.682,148.795
C02583=1148.476,235.359,-65.988,-177.690,7.685,148.795
C02584=1148.471,235.631,-66.016,-177.687,7.689,148.795
C02585=1148.466,235.903,-66.045,-177.684,7.691,148.795
C02586=1148.462,236.175,-66.074,-177.681,7.694,148.795
C02587=1148.457,236.424,-66.100,-177.678,7.697,148.795
C02588=1148.453,236.672,-66.127,-177.675,7.700,148.795
C02589=1148.449,236.921,-66.154,-177.673,7.703,148.795
C02590=1148.444,237.170,-66.180,-177.670,7.705,148.794
C02591=1148.440,237.418,-66.207,-177.668,7.708,148.794
C02592=1148.435,237.666,-66.234,-177.665,7.711,148.794
C02593=1148.431,237.915,-66.260,-177.662,7.713,148.794
C02594=1148.426,238.164,-66.287,-177.659,7.716,148.794
C02595=1148.422,238.412,-66.313,-177.656,7.719,148.794
C02596=1148.418,238.660,-66.340,-177.653,7.722,148.794
C02597=1148.413,238.909,-66.367,-177.651,7.724,148.794
C02598=1148.409,239.158,-66.393,-177.648,7.727,148.794
C02599=1148.404,239.406,-66.420,-177.645,7.730,148.793
C02600=1148.399,239.655,-66.447,-177.643,7.733,148.793
C02601=1148.396,239.903,-66.474,-177.640,7.736,148.793
C02602=1148.391,240.151,-66.501,-177.637,7.739,148.793
C02603=1148.386,240.401,-66.527,-177.634,7.741,148.793
C02604=1148.382,240.649,-66.553,-177.631,7.744,148.793
C02605=1148.377,240.897,-66.581,-177.629,7.746,148.793
C02606=1148.373,241.146,-66.608,-177.626,7.749,148.793
C02607=1148.369,241.394,-66.634,-177.623,7.752,148.793
C02608=1148.364,241.642,-66.661,-177.620,7.755,148.793
C02609=1148.359,241.891,-66.688,-177.618,7.758,148.792
C02610=1148.356,242.139,-66.715,-177.615,7.761,148.792
C02611=1148.351,242.388,-66.742,-177.612,7.764,148.792
C02612=1148.347,242.637,-66.769,-177.609,7.767,148.792
C02613=1148.342,242.885,-66.796,-177.607,7.770,148.792
C02614=1148.338,243.133,-66.823,-177.604,7.772,148.792
C02615=1148.334,243.382,-66.850,-177.601,7.775,148.792
C02616=1148.329,243.630,-66.877,-177.598,7.778,148.792
C02617=1148.324,243.879,-66.904,-177.596,7.780,148.792
C02618=1148.320,244.127,-66.930,-177.593,7.783,148.792
C02619=1148.316,244.376,-66.958,-177.590,7.786,148.791
C02620=1148.312,244.625,-66.985,-177.587,7.789,148.791
C02621=1148.307,244.873,-67.012,-177.584,7.792,148.791
C02622=1148.302,245.122,-67.039,-177.582,7.795,148.791
C02623=1148.298,245.370,-67.066,-177.579,7.798,148.791
C02624=1148.294,245.618,-67.092,-177.576,7.801,148.791
C02625=1148.290,245.867,-67.121,-177.574,7.803,148.791
C02626=1148.285,246.116,-67.148,-177.571,7.806,148.791
C02627=1148.281,246.364,-67.175,-177.568,7.809,148.791
C02628=1148.276,246.613,-67.202,-177.565,7.812,148.791
C02629=1148.271,246.861,-67.229,-177.563,7.815,148.791
C02630=1148.268,247.110,-67.257,-177.560,7.818,148.791
C02631=1148.263,247.358,-67.284,-177.557,7.821,148.791
C02632=1148.259,247.606,-67.310,-177.554,7.824,148.791
C02633=1148.254,247.855,-67.338,-177.552,7.826,148.790
C02634=1148.250,248.103,-67.365,-177.549,7.829,148.790
C02635=1148.246,248.352,-67.393,-177.546,7.832,148.790
C02636=1148.241,248.600,-67.420,-177.543,7.835,148.790
C02637=1148.237,248.849,-67.447,-177.540,7.838,148.790
C02638=1148.232,249.097,-67.475,-177.538,7.840,148.790
C02639=1148.228,249.346,-67.502,-177.535,7.843,148.790
C02640=1148.224,249.594,-67.529,-177.533,7.846,148.790
C02641=1148.219,249.842,-67.557,-177.530,7.849,148.790
C02642=1148.215,250.091,-67.584,-177.527,7.852,148.790
C02643=1148.211,250.339,-67.612,-177.524,7.855,148.790
C02644=1148.206,250.588,-67.639,-177.521,7.858,148.790
C02645=1148.202,250.836,-67.666,-177.519,7.861,148.790
C02646=1148.198,251.085,-67.694,-177.516,7.864,148.789
C02647=1148.193,251.333,-67.721,-177.513,7.867,148.789
C02648=1148.189,251.581,-67.749,-177.510,7.870,148.789
C02649=1148.184,251.830,-67.776,-177.508,7.873,148.789
C02650=1148.180,252.078,-67.804,-177.505,7.875,148.789
C02651=1148.176,252.327,-67.832,-177.502,7.878,148.789
C02652=1148.171,252.575,-67.860,-177.499,7.881,148.789
C02653=1148.167,252.824,-67.887,-177.496,7.884,148.789
C02654=1148.162,253.072,-67.915,-177.494,7.887,148.789
C02655=1148.158,253.321,-67.942,-177.491,7.890,148.789
C02656=1148.154,253.569,-67.970,-177.488,7.893,148.789
C02657=1148.149,253.818,-67.997,-177.485,7.896,148.789
C02658=1148.145,254.066,-68.025,-177.483,7.899,148.789
C02659=1148.141,254.314,-68.053,-177.480,7.902,148.789
C02660=1148.136,254.563,-68.081,-177.478,7.904,148.788
C02661=1148.132,254.812,-68.109,-177.475,7.907,148.788
C02662=1148.127,255.060,-68.136,-177.472,7.910,148.788
C02663=1148.123,255.308,-68.164,-177.469,7.913,148.788
C02664=1148.119,255.556,-68.192,-177.466,7.916,148.788
C02665=1148.114,255.805,-68.220,-177.464,7.919,148.788
C02666=1148.110,256.054,-68.248,-177.461,7.922,148.788
C02667=1148.106,256.302,-68.276,-177.459,7.925,148.788
C02668=1148.101,256.550,-68.303,-177.456,7.928,148.788
C02669=1148.097,256.799,-68.331,-177.453,7.931,148.788
C02670=1148.092,257.047,-68.359,-177.450,7.934,148.788
C02671=1148.088,257.296,-68.387,-177.447,7.937,148.788
C02672=1148.084,257.543,-68.415,-177.445,7.939,148.788
C02673=1148.080,257.793,-68.443,-177.442,7.942,148.788
C02674=1148.075,258.041,-68.471,-177.439,7.945,148.788
C02675=1148.071,258.289,-68.499,-177.436,7.948,148.788
C02676=1148.067,258.537,-68.527,-177.433,7.951,148.788
C02677=1148.062,258.785,-68.555,-177.431,7.954,148.788
C02678=1148.058,259.034,-68.583,-177.428,7.957,148.788
C02679=1148.053,259.283,-68.610,-177.426,7.960,148.788
C02680=1148.049,259.531,-68.639,-177.423,7.963,148.788
C02681=1148.044,259.779,-68.667,-177.420,7.966,148.788
C02682=1148.041,260.028,-68.695,-177.417,7.969,148.788
C02683=1148.036,260.276,-68.723,-177.414,7.972,148.787
C02684=1148.032,260.525,-68.752,-177.412,7.975,148.787
C02685=1148.028,260.772,-68.779,-177.409,7.978,148.787
C02686=1148.023,261.021,-68.808,-177.406,7.981,148.787
C02687=1148.018,261.295,-68.839,-177.403,7.985,148.787
C02688=1148.014,261.568,-68.869,-177.400,7.988,148.787
C02689=1148.009,261.841,-68.901,-177.397,7.991,148.787
C02690=1148.004,262.114,-68.932,-177.394,7.994,148.787
C02691=1147.999,262.363,-68.961,-177.391,7.997,148.787
C02692=1147.995,262.611,-68.989,-177.389,8.000,148.787
C02693=1147.991,262.860,-69.017,-177.386,8.003,148.787
C02694=1147.986,263.108,-69.045,-177.383,8.006,148.787
C02695=1147.983,263.357,-69.073,-177.380,8.009,148.787
C02696=1147.978,263.605,-69.102,-177.378,8.012,148.787
C02697=1147.974,263.853,-69.130,-177.375,8.015,148.787
C02698=1147.969,264.102,-69.159,-177.372,8.018,148.787
C02699=1147.965,264.349,-69.187,-177.370,8.021,148.787
C02700=1147.961,264.598,-69.216,-177.367,8.024,148.787
C02701=1147.956,264.846,-69.244,-177.364,8.027,148.787
C02702=1147.952,265.095,-69.272,-177.361,8.030,148.787
C02703=1147.947,265.344,-69.301,-177.359,8.033,148.787
C02704=1147.943,265.591,-69.330,-177.356,8.036,148.787
C02705=1147.939,265.840,-69.358,-177.353,8.040,148.787
C02706=1147.934,266.088,-69.386,-177.350,8.043,148.787
C02707=1147.930,266.337,-69.415,-177.347,8.046,148.787
C02708=1147.927,266.585,-69.444,-177.345,8.049,148.787
C02709=1147.921,266.833,-69.472,-177.342,8.052,148.787
C02710=1147.917,267.082,-69.501,-177.339,8.055,148.787
C02711=1147.914,267.330,-69.530,-177.337,8.058,148.787
C02712=1147.908,267.578,-69.558,-177.334,8.061,148.787
C02713=1147.905,267.827,-69.586,-177.331,8.064,148.787
C02714=1147.900,268.075,-69.616,-177.328,8.067,148.787
C02715=1147.895,268.323,-69.644,-177.326,8.070,148.787
C02716=1147.892,268.572,-69.672,-177.323,8.073,148.787
C02717=1147.887,268.820,-69.702,-177.320,8.076,148.787
C02718=1147.882,269.068,-69.730,-177.318,8.079,148.787
C02719=1147.879,269.316,-69.759,-177.315,8.082,148.787
C02720=1147.874,269.565,-69.788,-177.313,8.085,148.787
C02721=1147.869,269.813,-69.816,-177.310,8.088,148.787
C02722=1147.865,270.061,-69.845,-177.306,8.092,148.787
C02723=1147.861,270.310,-69.873,-177.304,8.095,148.787
C02724=1147.857,270.558,-69.903,-177.301,8.098,148.787
C02725=1147.852,270.806,-69.931,-177.299,8.101,148.787
C02726=1147.848,271.055,-69.961,-177.296,8.104,148.787
C02727=1147.844,271.303,-69.989,-177.293,8.107,148.787
C02728=1147.839,271.551,-70.018,-177.291,8.110,148.787
C02729=1147.835,271.799,-70.047,-177.288,8.113,148.787
C02730=1147.831,272.048,-70.076,-177.285,8.116,148.787
C02731=1147.827,272.296,-70.105,-177.282,8.119,148.787
C02732=1147.822,272.544,-70.133,-177.280,8.122,148.787
C02733=1147.818,272.792,-70.163,-177.277,8.125,148.787
C02734=1147.814,273.041,-70.192,-177.274,8.128,148.787
C02735=1147.809,273.290,-70.221,-177.271,8.132,148.787
C02736=1147.806,273.538,-70.250,-177.269,8.135,148.787
C02737=1147.801,273.785,-70.279,-177.266,8.138,148.787
C02738=1147.797,274.034,-70.308,-177.263,8.141,148.787
C02739=1147.793,274.282,-70.337,-177.260,8.144,148.787
C02740=1147.788,274.531,-70.367,-177.258,8.147,148.787
C02741=1147.784,274.779,-70.395,-177.255,8.150,148.787
C02742=1147.779,275.027,-70.424,-177.253,8.153,148.787
C02743=1147.776,275.275,-70.453,-177.250,8.156,148.787
C02744=1147.771,275.523,-70.483,-177.247,8.159,148.787
C02745=1147.767,275.772,-70.512,-177.244,8.163,148.787
C02746=1147.763,276.020,-70.541,-177.241,8.166,148.787
C02747=1147.759,276.269,-70.570,-177.239,8.169,148.787
C02748=1147.754,276.516,-70.600,-177.236,8.172,148.787
C02749=1147.750,276.764,-70.629,-177.233,8.175,148.787
C02750=1147.745,277.013,-70.658,-177.231,8.178,148.787
C02751=1147.741,277.262,-70.687,-177.228,8.181,148.787
C02752=1147.737,277.510,-70.717,-177.226,8.184,148.787
C02753=1147.733,277.758,-70.746,-177.223,8.187,148.787
C02754=1147.728,278.006,-70.776,-177.220,8.191,148.787
C02755=1147.724,278.255,-70.805,-177.217,8.194,148.787
C02756=1147.719,278.502,-70.834,-177.215,8.197,148.787
C02757=1147.715,278.750,-70.864,-177.212,8.200,148.787
C02758=1147.711,278.999,-70.893,-177.209,8.203,148.787
C02759=1147.707,279.247,-70.922,-177.207,8.206,148.787
C02760=1147.703,279.495,-70.952,-177.204,8.209,148.787
C02761=1147.699,279.744,-70.981,-177.201,8.212,148.787
C02762=1147.694,279.992,-71.011,-177.198,8.216,148.787
C02763=1147.690,280.240,-71.040,-177.196,8.219,148.787
C02764=1147.686,280.488,-71.070,-177.193,8.222,148.787
C02765=1147.682,280.737,-71.099,-177.191,8.226,148.787
C02766=1147.678,280.985,-71.129,-177.188,8.228,148.787
C02767=1147.673,281.233,-71.158,-177.185,8.231,148.787
C02768=1147.669,281.482,-71.188,-177.183,8.235,148.787
C02769=1147.664,281.729,-71.217,-177.179,8.238,148.787
C02770=1147.660,281.977,-71.247,-177.177,8.242,148.787
C02771=1147.656,282.225,-71.277,-177.174,8.245,148.787
C02772=1147.651,282.473,-71.306,-177.171,8.248,148.787
C02773=1147.647,282.722,-71.336,-177.169,8.251,148.788
C02774=1147.642,282.970,-71.366,-177.166,8.254,148.788
C02775=1147.638,283.219,-71.395,-177.164,8.257,148.787
C02776=1147.634,283.466,-71.425,-177.161,8.261,148.788
C02777=1147.630,283.715,-71.455,-177.158,8.264,148.788
C02778=1147.626,283.963,-71.484,-177.156,8.267,148.788
C02779=1147.621,284.211,-71.514,-177.153,8.270,148.788
C02780=1147.617,284.459,-71.545,-177.150,8.273,148.788
C02781=1147.613,284.707,-71.574,-177.148,8.276,148.788
C02782=1147.609,284.956,-71.603,-177.144,8.280,148.788
C02783=1147.604,285.204,-71.634,-177.142,8.283,148.788
C02784=1147.601,285.452,-71.664,-177.139,8.286,148.788
C02785=1147.596,285.701,-71.693,-177.136,8.289,148.788
C02786=1147.593,285.948,-71.724,-177.134,8.292,148.788
C02787=1147.588,286.197,-71.754,-177.131,8.295,148.788
C02788=1147.583,286.445,-71.783,-177.128,8.299,148.788
C02789=1147.580,286.693,-71.813,-177.126,8.302,148.788
C02790=1147.575,286.941,-71.843,-177.123,8.306,148.788
C02791=1147.570,287.216,-71.877,-177.120,8.309,148.788
C02792=1147.566,287.492,-71.910,-177.117,8.312,148.788
C02793=1147.561,287.767,-71.943,-177.114,8.316,148.789
C02794=1147.556,288.042,-71.976,-177.111,8.320,148.789
C02795=1147.551,288.290,-72.006,-177.109,8.323,148.789
C02796=1147.548,288.539,-72.037,-177.106,8.326,148.789
C02797=1147.543,288.787,-72.067,-177.103,8.330,148.789
C02798=1147.539,289.035,-72.097,-177.101,8.333,148.789
C02799=1147.535,289.283,-72.127,-177.098,8.335,148.789
C02800=1147.531,289.531,-72.157,-177.095,8.340,148.789
C02801=1147.526,289.780,-72.187,-177.092,8.342,148.789
C02802=1147.522,290.027,-72.217,-177.090,8.346,148.789
C02803=1147.518,290.276,-72.247,-177.087,8.349,148.789
C02804=1147.514,290.524,-72.277,-177.085,8.352,148.789
C02805=1147.510,290.772,-72.308,-177.081,8.356,148.789
C02806=1147.506,291.020,-72.338,-177.079,8.359,148.789
C02807=1147.501,291.268,-72.368,-177.076,8.362,148.789
C02808=1147.497,291.516,-72.399,-177.074,8.365,148.790
C02809=1147.493,291.765,-72.429,-177.071,8.368,148.790
C02810=1147.489,292.013,-72.459,-177.068,8.372,148.790
C02811=1147.484,292.261,-72.490,-177.066,8.375,148.790
C02812=1147.480,292.509,-72.519,-177.063,8.378,148.790
C02813=1147.475,292.757,-72.550,-177.060,8.381,148.790
C02814=1147.472,293.005,-72.581,-177.058,8.385,148.790
C02815=1147.468,293.253,-72.611,-177.055,8.388,148.790
C02816=1147.463,293.502,-72.641,-177.052,8.392,148.790
C02817=1147.459,293.750,-72.672,-177.050,8.395,148.790
C02818=1147.456,293.998,-72.702,-177.047,8.398,148.790
C02819=1147.451,294.246,-72.733,-177.044,8.402,148.791
C02820=1147.446,294.494,-72.764,-177.042,8.405,148.790
C02821=1147.442,294.741,-72.794,-177.039,8.408,148.791
C02822=1147.438,294.991,-72.824,-177.037,8.411,148.791
C02823=1147.434,295.238,-72.855,-177.034,8.415,148.791
C02824=1147.430,295.486,-72.885,-177.031,8.418,148.791
C02825=1147.425,295.734,-72.916,-177.029,8.421,148.791
C02826=1147.422,295.983,-72.947,-177.026,8.424,148.791
C02827=1147.417,296.231,-72.977,-177.023,8.428,148.791
C02828=1147.413,296.479,-73.008,-177.021,8.432,148.791
C02829=1147.409,296.727,-73.039,-177.018,8.435,148.791
C02830=1147.405,296.975,-73.069,-177.015,8.438,148.791
C02831=1147.400,297.223,-73.100,-177.013,8.441,148.791
C02832=1147.396,297.470,-73.130,-177.010,8.445,148.792
C02833=1147.392,297.719,-73.161,-177.007,8.448,148.792
C02834=1147.388,297.967,-73.192,-177.005,8.451,148.792
C02835=1147.384,298.215,-73.222,-177.002,8.454,148.792
C02836=1147.380,298.463,-73.254,-176.999,8.458,148.792
C02837=1147.375,298.711,-73.284,-176.997,8.461,148.792
C02838=1147.370,298.959,-73.315,-176.994,8.465,148.792
C02839=1147.367,299.208,-73.346,-176.992,8.468,148.792
C02840=1147.363,299.456,-73.376,-176.989,8.472,148.792
C02841=1147.358,299.703,-73.408,-176.986,8.475,148.792
C02842=1147.354,299.952,-73.439,-176.984,8.478,148.793
C02843=1147.350,300.199,-73.469,-176.981,8.481,148.793
C02844=1147.346,300.448,-73.500,-176.978,8.485,148.793
C02845=1147.342,300.696,-73.531,-176.976,8.488,148.793
C02846=1147.337,300.944,-73.562,-176.973,8.491,148.793
C02847=1147.333,301.192,-73.594,-176.970,8.495,148.793
C02848=1147.329,301.440,-73.624,-176.968,8.499,148.793
C02849=1147.325,301.687,-73.655,-176.965,8.501,148.793
C02850=1147.321,301.936,-73.686,-176.962,8.505,148.793
C02851=1147.317,302.183,-73.717,-176.960,8.509,148.794
C02852=1147.313,302.432,-73.748,-176.957,8.512,148.794
C02853=1147.308,302.680,-73.779,-176.954,8.515,148.794
C02854=1147.304,302.927,-73.811,-176.952,8.518,148.794
C02855=1147.300,303.176,-73.842,-176.949,8.522,148.794
C02856=1147.295,303.424,-73.872,-176.946,8.525,148.794
C02857=1147.291,303.672,-73.904,-176.944,8.529,148.794
C02858=1147.287,303.920,-73.935,-176.941,8.532,148.794
C02859=1147.283,304.168,-73.966,-176.938,8.536,148.795
C02860=1147.279,304.416,-73.997,-176.936,8.539,148.795
C02861=1147.275,304.664,-74.028,-176.933,8.542,148.795
C02862=1147.271,304.912,-74.060,-176.930,8.546,148.795
C02863=1147.266,305.160,-74.090,-176.928,8.549,148.795
C02864=1147.262,305.408,-74.122,-176.926,8.552,148.795
C02865=1147.258,305.656,-74.153,-176.922,8.556,148.795
C02866=1147.254,305.904,-74.184,-176.920,8.559,148.795
C02867=1147.250,306.152,-74.216,-176.918,8.563,148.796
C02868=1147.246,306.400,-74.247,-176.914,8.567,148.796
C02869=1147.241,306.648,-74.278,-176.912,8.570,148.796
C02870=1147.238,306.896,-74.310,-176.910,8.573,148.796
C02871=1147.232,307.144,-74.341,-176.907,8.576,148.796
C02872=1147.228,307.392,-74.373,-176.904,8.580,148.796
C02873=1147.224,307.640,-74.404,-176.902,8.583,148.796
C02874=1147.220,307.888,-74.436,-176.899,8.587,148.797
C02875=1147.216,308.137,-74.467,-176.896,8.590,148.797
C02876=1147.212,308.384,-74.499,-176.894,8.594,148.797
C02877=1147.208,308.632,-74.530,-176.891,8.597,148.797
C02878=1147.203,308.880,-74.561,-176.889,8.601,148.797
C02879=1147.200,309.128,-74.593,-176.886,8.604,148.797
C02880=1147.195,309.375,-74.624,-176.883,8.607,148.797
C02881=1147.191,309.624,-74.656,-176.881,8.611,148.798
C02882=1147.186,309.872,-74.688,-176.878,8.615,148.798
C02883=1147.183,310.120,-74.720,-176.876,8.618,148.798
C02884=1147.179,310.368,-74.751,-176.873,8.622,148.798
C02885=1147.174,310.616,-74.782,-176.870,8.625,148.798
C02886=1147.171,310.864,-74.814,-176.868,8.628,148.798
C02887=1147.166,311.111,-74.845,-176.865,8.632,148.799
C02888=1147.162,311.359,-74.878,-176.862,8.635,148.799
C02889=1147.158,311.608,-74.910,-176.860,8.638,148.799
C02890=1147.154,311.855,-74.941,-176.857,8.642,148.799
C02891=1147.150,312.104,-74.972,-176.855,8.646,148.799
C02892=1147.145,312.352,-75.005,-176.852,8.649,148.799
C02893=1147.141,312.599,-75.036,-176.849,8.653,148.799
C02894=1147.137,312.847,-75.068,-176.847,8.656,148.799
C02895=1147.133,313.125,-75.104,-176.844,8.660,148.800
C02896=1147.128,313.403,-75.139,-176.841,8.664,148.800
C02897=1147.123,313.681,-75.175,-176.838,8.667,148.800
C02898=1147.119,313.958,-75.210,-176.835,8.671,148.800
C02899=1147.114,314.206,-75.243,-176.832,8.675,148.800
C02900=1147.110,314.454,-75.274,-176.830,8.679,148.801
C02901=1147.107,314.702,-75.306,-176.828,8.682,148.801
C02902=1147.102,314.949,-75.338,-176.825,8.686,148.801
C02903=1147.098,315.198,-75.370,-176.822,8.689,148.801
C02904=1147.094,315.446,-75.402,-176.819,8.693,148.801
C02905=1147.090,315.693,-75.433,-176.817,8.696,148.801
C02906=1147.085,315.941,-75.466,-176.814,8.700,148.802
C02907=1147.082,316.189,-75.498,-176.811,8.704,148.802
C02908=1147.077,316.438,-75.530,-176.809,8.707,148.802
C02909=1147.073,316.685,-75.562,-176.807,8.710,148.802
C02910=1147.070,316.933,-75.594,-176.804,8.714,148.802
C02911=1147.065,317.181,-75.627,-176.802,8.717,148.803
C02912=1147.061,317.429,-75.658,-176.799,8.720,148.803
C02913=1147.056,317.677,-75.691,-176.796,8.725,148.803
C02914=1147.053,317.925,-75.722,-176.794,8.728,148.803
C02915=1147.049,318.172,-75.755,-176.791,8.732,148.803
C02916=1147.045,318.420,-75.787,-176.788,8.735,148.803
C02917=1147.041,318.668,-75.819,-176.786,8.738,148.804
C02918=1147.036,318.916,-75.851,-176.783,8.743,148.804
C02919=1147.032,319.164,-75.883,-176.781,8.746,148.804
C02920=1147.028,319.412,-75.916,-176.778,8.749,148.804
C02921=1147.025,319.660,-75.948,-176.775,8.753,148.804
C02922=1147.020,319.908,-75.980,-176.773,8.756,148.805
C02923=1147.016,320.155,-76.013,-176.770,8.760,148.805
C02924=1147.012,320.403,-76.045,-176.767,8.763,148.805
C02925=1147.008,320.651,-76.077,-176.765,8.767,148.805
C02926=1147.004,320.899,-76.110,-176.762,8.771,148.805
C02927=1147.000,321.147,-76.142,-176.760,8.774,148.805
C02928=1146.995,321.395,-76.174,-176.757,8.778,148.806
C02929=1146.992,321.642,-76.207,-176.755,8.781,148.806
C02930=1146.987,321.891,-76.239,-176.752,8.785,148.806
C02931=1146.983,322.138,-76.272,-176.749,8.789,148.806
C02932=1146.979,322.386,-76.304,-176.747,8.792,148.806
C02933=1146.975,322.634,-76.337,-176.744,8.796,148.807
C02934=1146.972,322.882,-76.369,-176.742,8.799,148.807
C02935=1146.966,323.130,-76.401,-176.740,8.803,148.807
C02936=1146.963,323.377,-76.434,-176.737,8.807,148.807
C02937=1146.959,323.625,-76.467,-176.734,8.810,148.807
C02938=1146.955,323.873,-76.499,-176.731,8.814,148.808
C02939=1146.951,324.121,-76.532,-176.729,8.817,148.808
C02940=1146.947,324.369,-76.564,-176.726,8.821,148.808
C02941=1146.943,324.617,-76.598,-176.724,8.825,148.808
C02942=1146.939,324.865,-76.629,-176.721,8.828,148.809
C02943=1146.935,325.112,-76.663,-176.719,8.832,148.809
C02944=1146.930,325.361,-76.695,-176.716,8.835,148.809
C02945=1146.927,325.608,-76.728,-176.713,8.839,148.809
C02946=1146.923,325.856,-76.761,-176.711,8.843,148.809
C02947=1146.918,326.104,-76.793,-176.708,8.847,148.810
C02948=1146.914,326.351,-76.826,-176.706,8.850,148.810
C02949=1146.910,326.599,-76.859,-176.703,8.853,148.810
C02950=1146.906,326.847,-76.891,-176.701,8.857,148.810
C02951=1146.902,327.095,-76.924,-176.698,8.861,148.810
C02952=1146.897,327.343,-76.957,-176.695,8.865,148.811
C02953=1146.894,327.590,-76.990,-176.693,8.868,148.811
C02954=1146.890,327.838,-77.022,-176.690,8.872,148.811
C02955=1146.885,328.086,-77.055,-176.688,8.875,148.811
C02956=1146.881,328.334,-77.089,-176.685,8.879,148.811
C02957=1146.877,328.582,-77.122,-176.682,8.883,148.812
C02958=1146.873,328.829,-77.155,-176.680,8.886,148.812
C02959=1146.869,329.077,-77.187,-176.677,8.890,148.812
C02960=1146.865,329.325,-77.220,-176.675,8.893,148.812
C02961=1146.861,329.573,-77.253,-176.672,8.897,148.813
C02962=1146.857,329.821,-77.286,-176.670,8.901,148.813
C02963=1146.853,330.068,-77.319,-176.667,8.905,148.813
C02964=1146.849,330.316,-77.353,-176.665,8.908,148.813
C02965=1146.844,330.564,-77.386,-176.662,8.912,148.814
C02966=1146.840,330.811,-77.419,-176.660,8.916,148.814
C02967=1146.837,331.059,-77.451,-176.657,8.920,148.814
C02968=1146.832,331.307,-77.484,-176.654,8.923,148.814
C02969=1146.828,331.555,-77.517,-176.652,8.926,148.814
C02970=1146.825,331.803,-77.551,-176.649,8.930,148.815
C02971=1146.821,332.051,-77.584,-176.647,8.934,148.815
C02972=1146.817,332.299,-77.617,-176.644,8.938,148.815
C02973=1146.812,332.547,-77.650,-176.642,8.941,148.816
C02974=1146.809,332.794,-77.684,-176.639,8.945,148.816
C02975=1146.804,333.041,-77.717,-176.637,8.949,148.816
C02976=1146.800,333.289,-77.750,-176.634,8.953,148.816
C02977=1146.796,333.537,-77.783,-176.631,8.956,148.816
C02978=1146.792,333.785,-77.816,-176.629,8.960,148.817
C02979=1146.788,334.032,-77.850,-176.626,8.963,148.817
C02980=1146.784,334.281,-77.883,-176.623,8.967,148.817
C02981=1146.780,334.528,-77.916,-176.621,8.971,148.817
C02982=1146.776,334.776,-77.949,-176.619,8.975,148.818
C02983=1146.772,335.023,-77.983,-176.616,8.978,148.818
C02984=1146.768,335.271,-78.016,-176.613,8.982,148.818
C02985=1146.764,335.519,-78.050,-176.611,8.986,148.818
C02986=1146.760,335.766,-78.083,-176.608,8.990,148.819
C02987=1146.756,336.015,-78.117,-176.606,8.993,148.819
C02988=1146.752,336.262,-78.151,-176.603,8.997,148.819
C02989=1146.748,336.510,-78.184,-176.601,9.001,148.819
C02990=1146.743,336.758,-78.217,-176.598,9.005,148.820
C02991=1146.740,337.005,-78.251,-176.596,9.008,148.820
C02992=1146.735,337.253,-78.284,-176.593,9.012,148.820
C02993=1146.732,337.501,-78.318,-176.591,9.016,148.821
C02994=1146.728,337.748,-78.352,-176.588,9.020,148.821
C02995=1146.723,337.996,-78.385,-176.586,9.023,148.821
C02996=1146.719,338.244,-78.418,-176.583,9.027,148.821
C02997=1146.715,338.491,-78.452,-176.580,9.030,148.821
C02998=1146.712,338.739,-78.486,-176.578,9.035,148.822
C02999=1146.706,339.019,-78.524,-176.575,9.039,148.822
C03000=1146.702,339.300,-78.562,-176.572,9.043,148.822
C03001=1146.698,339.580,-78.600,-176.569,9.047,148.823
C03002=1146.694,339.861,-78.638,-176.567,9.052,148.823
C03003=1146.689,340.109,-78.672,-176.564,9.056,148.823
C03004=1146.685,340.356,-78.706,-176.561,9.059,148.824
C03005=1146.681,340.604,-78.739,-176.559,9.063,148.824
C03006=1146.678,340.851,-78.773,-176.557,9.067,148.824
C03007=1146.673,341.099,-78.807,-176.554,9.071,148.824
C03008=1146.669,341.346,-78.841,-176.551,9.074,148.825
C03009=1146.665,341.595,-78.874,-176.548,9.078,148.825
C03010=1146.661,341.842,-78.909,-176.547,9.082,148.825
C03011=1146.657,342.089,-78.943,-176.544,9.086,148.826
C03012=1146.653,342.337,-78.976,-176.541,9.090,148.826
C03013=1146.649,342.585,-79.011,-176.538,9.093,148.826
C03014=1146.645,342.832,-79.045,-176.536,9.097,148.826
C03015=1146.641,343.080,-79.078,-176.534,9.101,148.827
C03016=1146.637,343.328,-79.113,-176.531,9.105,148.827
C03017=1146.633,343.575,-79.146,-176.528,9.108,148.827
C03018=1146.628,343.823,-79.180,-176.526,9.112,148.828
C03019=1146.625,344.071,-79.214,-176.524,9.116,148.828
C03020=1146.621,344.318,-79.248,-176.521,9.120,148.828
C03021=1146.616,344.566,-79.282,-176.518,9.124,148.828
C03022=1146.613,344.814,-79.316,-176.516,9.127,148.829
C03023=1146.608,345.062,-79.351,-176.513,9.132,148.829
C03024=1146.605,345.309,-79.385,-176.511,9.135,148.829
C03025=1146.600,345.557,-79.419,-176.508,9.139,148.830
C03026=1146.596,345.804,-79.453,-176.506,9.142,148.830
C03027=1146.593,346.052,-79.486,-176.503,9.147,148.830
C03028=1146.589,346.300,-79.521,-176.501,9.150,148.830
C03029=1146.585,346.547,-79.555,-176.498,9.154,148.831
C03030=1146.581,346.795,-79.590,-176.495,9.158,148.831
C03031=1146.577,347.042,-79.624,-176.493,9.162,148.831
C03032=1146.572,347.290,-79.658,-176.490,9.166,148.832
C03033=1146.569,347.538,-79.692,-176.488,9.169,148.832
C03034=1146.564,347.785,-79.726,-176.485,9.174,148.832
C03035=1146.560,348.033,-79.761,-176.483,9.178,148.832
C03036=1146.557,348.281,-79.795,-176.480,9.181,148.833
C03037=1146.553,348.529,-79.830,-176.478,9.185,148.833
C03038=1146.549,348.776,-79.864,-176.475,9.189,148.833
C03039=1146.544,349.023,-79.898,-176.473,9.193,148.834
C03040=1146.541,349.271,-79.932,-176.471,9.196,148.834
C03041=1146.536,349.518,-79.967,-176.468,9.200,148.834
C03042=1146.532,349.767,-80.002,-176.465,9.205,148.835
C03043=1146.529,350.014,-80.036,-176.463,9.208,148.835
C03044=1146.525,350.262,-80.070,-176.460,9.212,148.835
C03045=1146.521,350.508,-80.105,-176.458,9.216,148.836
C03046=1146.517,350.756,-80.140,-176.455,9.220,148.836
C03047=1146.513,351.004,-80.174,-176.453,9.224,148.836
C03048=1146.509,351.252,-80.209,-176.450,9.227,148.836
C03049=1146.505,351.499,-80.243,-176.447,9.232,148.837
C03050=1146.501,351.747,-80.278,-176.445,9.235,148.837
C03051=1146.497,351.994,-80.312,-176.443,9.239,148.837
C03052=1146.493,352.242,-80.347,-176.440,9.244,148.838
C03053=1146.489,352.489,-80.382,-176.438,9.247,148.838
C03054=1146.485,352.737,-80.416,-176.435,9.251,148.838
C03055=1146.481,352.984,-80.450,-176.432,9.255,148.839
C03056=1146.477,353.232,-80.486,-176.430,9.259,148.839
C03057=1146.473,353.479,-80.520,-176.428,9.263,148.839
C03058=1146.469,353.727,-80.555,-176.425,9.266,148.840
C03059=1146.465,353.975,-80.590,-176.422,9.270,148.840
C03060=1146.461,354.222,-80.625,-176.420,9.275,148.840
C03061=1146.457,354.470,-80.660,-176.417,9.278,148.841
C03062=1146.453,354.717,-80.693,-176.415,9.282,148.841
C03063=1146.450,354.965,-80.729,-176.412,9.286,148.841
C03064=1146.445,355.212,-80.763,-176.410,9.290,148.842
C03065=1146.442,355.460,-80.799,-176.407,9.294,148.842
C03066=1146.438,355.708,-80.833,-176.405,9.297,148.842
C03067=1146.434,355.955,-80.868,-176.402,9.302,148.843
C03068=1146.430,356.202,-80.903,-176.399,9.306,148.843
C03069=1146.426,356.451,-80.938,-176.398,9.309,148.843
C03070=1146.422,356.697,-80.973,-176.395,9.314,148.844
C03071=1146.418,356.945,-81.008,-176.392,9.318,148.844
C03072=1146.414,357.192,-81.043,-176.390,9.321,148.844
C03073=1146.410,357.440,-81.078,-176.387,9.326,148.845
C03074=1146.407,357.688,-81.113,-176.384,9.330,148.845
C03075=1146.402,357.935,-81.148,-176.383,9.333,148.845
C03076=1146.398,358.183,-81.183,-176.380,9.337,148.846
C03077=1146.395,358.430,-81.219,-176.377,9.342,148.846
C03078=1146.390,358.677,-81.253,-176.375,9.345,148.846
C03079=1146.387,358.925,-81.289,-176.372,9.349,148.847
C03080=1146.383,359.173,-81.323,-176.369,9.353,148.847
C03081=1146.378,359.420,-81.359,-176.367,9.357,148.847
C03082=1146.375,359.667,-81.394,-176.365,9.361,148.848
C03083=1146.371,359.915,-81.429,-176.362,9.365,148.848
C03084=1146.367,360.163,-81.465,-176.360,9.369,148.848
C03085=1146.364,360.409,-81.499,-176.357,9.373,148.849
C03086=1146.360,360.658,-81.534,-176.354,9.377,148.849
C03087=1146.356,360.905,-81.570,-176.351,9.381,148.849
C03088=1146.352,361.152,-81.605,-176.349,9.385,148.850
C03089=1146.348,361.399,-81.640,-176.347,9.389,148.850
C03090=1146.343,361.648,-81.676,-176.344,9.393,148.850
C03091=1146.340,361.895,-81.711,-176.341,9.397,148.851
C03092=1146.335,362.142,-81.746,-176.339,9.401,148.851
C03093=1146.332,362.390,-81.782,-176.336,9.405,148.851
C03094=1146.328,362.637,-81.818,-176.333,9.409,148.852
C03095=1146.324,362.885,-81.853,-176.331,9.414,148.852
C03096=1146.320,363.133,-81.888,-176.328,9.418,148.852
C03097=1146.316,363.380,-81.923,-176.326,9.421,148.853
C03098=1146.312,363.627,-81.959,-176.323,9.425,148.853
C03099=1146.309,363.875,-81.994,-176.321,9.430,148.854
C03100=1146.305,364.122,-82.030,-176.318,9.434,148.854
C03101=1146.301,364.370,-82.065,-176.315,9.438,148.854
C03102=1146.297,364.616,-82.100,-176.313,9.441,148.855
C03103=1146.293,364.900,-82.141,-176.310,9.447,148.855
C03104=1146.288,365.183,-82.182,-176.306,9.452,148.855
C03105=1146.284,365.466,-82.223,-176.304,9.456,148.856
C03106=1146.280,365.750,-82.264,-176.300,9.461,148.856
C03107=1146.275,365.998,-82.300,-176.298,9.464,148.857
C03108=1146.271,366.245,-82.335,-176.296,9.469,148.857
C03109=1146.268,366.493,-82.371,-176.293,9.473,148.857
C03110=1146.264,366.740,-82.406,-176.290,9.477,148.858
C03111=1146.260,366.988,-82.443,-176.288,9.481,148.858
C03112=1146.255,367.235,-82.478,-176.285,9.486,148.858
C03113=1146.252,367.482,-82.513,-176.282,9.490,148.859
C03114=1146.248,367.730,-82.549,-176.280,9.494,148.859
C03115=1146.244,367.977,-82.586,-176.277,9.498,148.859
C03116=1146.240,368.224,-82.621,-176.275,9.502,148.860
C03117=1146.237,368.472,-82.657,-176.272,9.506,148.860
C03118=1146.232,368.720,-82.693,-176.269,9.510,148.861
C03119=1146.229,368.967,-82.728,-176.267,9.515,148.861
C03120=1146.225,369.214,-82.765,-176.264,9.519,148.861
C03121=1146.221,369.461,-82.800,-176.262,9.523,148.862
C03122=1146.217,369.709,-82.836,-176.260,9.527,148.862
C03123=1146.213,369.956,-82.872,-176.257,9.531,148.863
C03124=1146.209,370.203,-82.908,-176.254,9.535,148.863
C03125=1146.205,370.451,-82.944,-176.252,9.540,148.863
C03126=1146.202,370.698,-82.980,-176.249,9.544,148.864
C03127=1146.197,370.946,-83.016,-176.246,9.548,148.864
C03128=1146.194,371.193,-83.052,-176.244,9.553,148.865
C03129=1146.190,371.440,-83.088,-176.242,9.556,148.865
C03130=1146.186,371.688,-83.124,-176.239,9.560,148.865
C03131=1146.182,371.935,-83.160,-176.236,9.565,148.866
C03132=1146.178,372.183,-83.197,-176.234,9.569,148.866
C03133=1146.175,372.430,-83.232,-176.231,9.573,148.867
C03134=1146.171,372.677,-83.269,-176.230,9.577,148.867
C03135=1146.167,372.925,-83.305,-176.227,9.581,148.868
C03136=1146.164,373.172,-83.341,-176.225,9.586,148.868
C03137=1146.159,373.419,-83.377,-176.222,9.590,148.869
C03138=1146.156,373.666,-83.413,-176.220,9.595,148.869
C03139=1146.151,373.914,-83.450,-176.218,9.598,148.869
C03140=1146.148,374.161,-83.486,-176.215,9.603,148.870
C03141=1146.144,374.408,-83.523,-176.213,9.607,148.870
C03142=1146.140,374.656,-83.558,-176.211,9.610,148.871
C03143=1146.136,374.903,-83.595,-176.208,9.615,148.871
C03144=1146.132,375.151,-83.631,-176.206,9.619,148.872
C03145=1146.128,375.398,-83.667,-176.204,9.623,148.872
C03146=1146.124,375.645,-83.704,-176.202,9.628,148.873
C03147=1146.121,375.892,-83.740,-176.200,9.631,148.873
C03148=1146.117,376.139,-83.777,-176.197,9.635,148.874
C03149=1146.114,376.387,-83.813,-176.195,9.640,148.874
C03150=1146.109,376.635,-83.849,-176.193,9.644,148.875
C03151=1146.105,376.882,-83.886,-176.191,9.648,148.875
C03152=1146.102,377.129,-83.923,-176.189,9.652,148.876
C03153=1146.098,377.377,-83.959,-176.187,9.656,148.876
C03154=1146.094,377.624,-83.995,-176.185,9.660,148.877
C03155=1146.090,377.871,-84.032,-176.183,9.664,148.877
C03156=1146.086,378.118,-84.069,-176.181,9.669,148.878
C03157=1146.083,378.365,-84.105,-176.179,9.672,148.879
C03158=1146.078,378.613,-84.141,-176.178,9.676,148.879
C03159=1146.074,378.860,-84.178,-176.177,9.680,148.880
C03160=1146.071,379.107,-84.215,-176.174,9.684,148.880
C03161=1146.067,379.355,-84.251,-176.173,9.688,148.881
C03162=1146.063,379.602,-84.288,-176.171,9.692,148.881
C03163=1146.060,379.849,-84.325,-176.170,9.696,148.882
C03164=1146.055,380.097,-84.361,-176.168,9.700,148.883
C03165=1146.051,380.344,-84.398,-176.167,9.704,148.883
C03166=1146.047,380.591,-84.434,-176.165,9.708,148.884
C03167=1146.044,380.838,-84.471,-176.164,9.712,148.885
C03168=1146.040,381.086,-84.508,-176.162,9.715,148.885
C03169=1146.036,381.333,-84.545,-176.161,9.719,148.886
C03170=1146.033,381.580,-84.581,-176.159,9.723,148.886
C03171=1146.029,381.827,-84.618,-176.159,9.727,148.887
C03172=1146.025,382.074,-84.655,-176.157,9.730,148.888
C03173=1146.021,382.322,-84.692,-176.156,9.734,148.888
C03174=1146.018,382.569,-84.728,-176.155,9.738,148.889
C03175=1146.014,382.816,-84.765,-176.154,9.742,148.890
C03176=1146.010,383.063,-84.802,-176.153,9.745,148.890
C03177=1146.006,383.310,-84.839,-176.152,9.748,148.891
C03178=1146.002,383.558,-84.876,-176.151,9.752,148.892
C03179=1145.999,383.805,-84.912,-176.151,9.756,148.893
C03180=1145.995,384.052,-84.949,-176.150,9.759,148.893
C03181=1145.991,384.300,-84.986,-176.149,9.762,148.894
C03182=1145.986,384.547,-85.023,-176.149,9.765,148.895
C03183=1145.983,384.795,-85.060,-176.148,9.769,148.895
C03184=1145.980,385.042,-85.096,-176.148,9.772,148.896
C03185=1145.976,385.289,-85.133,-176.147,9.776,148.897
C03186=1145.971,385.536,-85.170,-176.147,9.779,148.898
C03187=1145.968,385.783,-85.208,-176.146,9.782,148.898
C03188=1145.964,386.030,-85.245,-176.146,9.785,148.899
C03189=1145.960,386.278,-85.282,-176.146,9.788,148.900
C03190=1145.957,386.524,-85.318,-176.146,9.791,148.901
C03191=1145.953,386.772,-85.355,-176.146,9.794,148.902
C03192=1145.949,387.020,-85.392,-176.146,9.797,148.902
C03193=1145.945,387.267,-85.429,-176.146,9.800,148.903
C03194=1145.941,387.514,-85.466,-176.146,9.803,148.904
C03195=1145.937,387.761,-85.503,-176.146,9.806,148.905
C03196=1145.934,388.008,-85.541,-176.146,9.808,148.905
C03197=1145.930,388.255,-85.577,-176.146,9.812,148.906
C03198=1145.926,388.502,-85.614,-176.146,9.815,148.907
C03199=1145.922,388.750,-85.651,-176.147,9.818,148.908
C03200=1145.919,388.998,-85.688,-176.147,9.820,148.909
C03201=1145.915,389.244,-85.725,-176.147,9.823,148.909
C03202=1145.911,389.491,-85.762,-176.148,9.826,148.910
C03203=1145.907,389.738,-85.799,-176.148,9.828,148.911
C03204=1145.904,389.986,-85.836,-176.149,9.830,148.912
C03205=1145.900,390.233,-85.873,-176.150,9.833,148.913
C03206=1145.896,390.480,-85.909,-176.150,9.836,148.913
C03207=1145.891,390.767,-85.953,-176.151,9.839,148.915
C03208=1145.887,391.054,-85.996,-176.151,9.842,148.915
C03209=1145.883,391.341,-86.039,-176.152,9.845,148.916
C03210=1145.878,391.628,-86.082,-176.153,9.848,148.917
C03211=1145.874,391.876,-86.119,-176.154,9.850,148.918
C03212=1145.871,392.122,-86.155,-176.154,9.853,148.919
C03213=1145.867,392.369,-86.193,-176.155,9.855,148.920
C03214=1145.863,392.616,-86.230,-176.156,9.858,148.921
C03215=1145.860,392.864,-86.267,-176.157,9.860,148.922
C03216=1145.855,393.111,-86.304,-176.158,9.862,148.922
C03217=1145.852,393.358,-86.341,-176.158,9.865,148.923
C03218=1145.848,393.605,-86.378,-176.159,9.867,148.924
C03219=1145.844,393.853,-86.416,-176.160,9.869,148.925
C03220=1145.840,394.100,-86.452,-176.161,9.872,148.926
C03221=1145.836,394.347,-86.489,-176.162,9.874,148.927
C03222=1145.833,394.594,-86.526,-176.163,9.876,148.927
C03223=1145.829,394.841,-86.563,-176.164,9.877,148.928
C03224=1145.825,395.089,-86.600,-176.165,9.880,148.929
C03225=1145.821,395.336,-86.637,-176.165,9.882,148.930
C03226=1145.818,395.583,-86.675,-176.167,9.884,148.931
C03227=1145.814,395.830,-86.712,-176.168,9.887,148.932
C03228=1145.810,396.077,-86.749,-176.169,9.889,148.932
C03229=1145.806,396.325,-86.786,-176.170,9.891,148.933
C03230=1145.802,396.573,-86.823,-176.171,9.893,148.934
C03231=1145.798,396.819,-86.861,-176.172,9.895,148.935
C03232=1145.794,397.066,-86.897,-176.173,9.897,148.936
C03233=1145.790,397.313,-86.934,-176.174,9.899,148.937
C03234=1145.787,397.561,-86.971,-176.175,9.901,148.937
C03235=1145.784,397.808,-87.008,-176.176,9.903,148.938
C03236=1145.780,398.055,-87.045,-176.178,9.905,148.939
C03237=1145.776,398.302,-87.082,-176.179,9.907,148.940
C03238=1145.772,398.550,-87.119,-176.180,9.909,148.941
C03239=1145.768,398.797,-87.156,-176.181,9.911,148.942
C03240=1145.764,399.044,-87.194,-176.182,9.913,148.942
C03241=1145.760,399.291,-87.231,-176.183,9.915,148.943
C03242=1145.757,399.539,-87.268,-176.184,9.917,148.944
C03243=1145.752,399.786,-87.305,-176.185,9.919,148.945
C03244=1145.749,400.033,-87.342,-176.186,9.922,148.946
C03245=1145.745,400.280,-87.380,-176.188,9.923,148.947
C03246=1145.742,400.527,-87.416,-176.189,9.925,148.947
C03247=1145.738,400.774,-87.453,-176.190,9.927,148.948
C03248=1145.734,401.021,-87.490,-176.191,9.929,148.949
C03249=1145.730,401.269,-87.527,-176.192,9.931,148.950
C03250=1145.726,401.516,-87.564,-176.194,9.933,148.951
C03251=1145.722,401.763,-87.601,-176.195,9.935,148.952
C03252=1145.718,402.011,-87.638,-176.196,9.937,148.952
C03253=1145.715,402.258,-87.676,-176.197,9.938,148.953
C03254=1145.711,402.505,-87.713,-176.198,9.940,148.954
C03255=1145.707,402.752,-87.750,-176.199,9.942,148.955
C03256=1145.703,402.999,-87.787,-176.200,9.944,148.955
C03257=1145.700,403.247,-87.824,-176.201,9.946,148.956
C03258=1145.696,403.494,-87.861,-176.202,9.948,148.957
C03259=1145.692,403.741,-87.898,-176.204,9.951,148.958
C03260=1145.688,403.988,-87.934,-176.205,9.952,148.959
C03261=1145.685,404.235,-87.972,-176.206,9.954,148.959
C03262=1145.681,404.482,-88.009,-176.207,9.956,148.960
C03263=1145.677,404.730,-88.046,-176.208,9.958,148.961
C03264=1145.673,404.977,-88.083,-176.209,9.960,148.962
C03265=1145.669,405.224,-88.121,-176.210,9.962,148.963
C03266=1145.665,405.471,-88.158,-176.211,9.964,148.964
C03267=1145.661,405.718,-88.195,-176.213,9.965,148.964
C03268=1145.658,405.966,-88.232,-176.214,9.967,148.965
C03269=1145.654,406.213,-88.269,-176.215,9.969,148.966
C03270=1145.650,406.460,-88.306,-176.216,9.971,148.967
C03271=1145.646,406.707,-88.343,-176.217,9.973,148.967
C03272=1145.643,406.955,-88.380,-176.218,9.975,148.968
C03273=1145.639,407.202,-88.417,-176.219,9.977,148.969
C03274=1145.635,407.449,-88.454,-176.219,9.979,148.970
C03275=1145.631,407.696,-88.491,-176.221,9.981,148.970
C03276=1145.627,407.944,-88.528,-176.222,9.983,148.971
C03277=1145.623,408.191,-88.565,-176.223,9.985,148.972
C03278=1145.620,408.437,-88.603,-176.223,9.987,148.973
C03279=1145.616,408.685,-88.640,-176.224,9.989,148.974
C03280=1145.612,408.932,-88.677,-176.225,9.990,148.974
C03281=1145.608,409.180,-88.714,-176.227,9.992,148.975
C03282=1145.605,409.427,-88.750,-176.228,9.994,148.976
C03283=1145.601,409.674,-88.788,-176.229,9.995,148.976
C03284=1145.597,409.921,-88.825,-176.230,9.998,148.977
C03285=1145.593,410.168,-88.862,-176.231,10.000,148.978
C03286=1145.589,410.415,-88.898,-176.231,10.002,148.979
C03287=1145.586,410.663,-88.936,-176.232,10.004,148.980
C03288=1145.582,410.910,-88.973,-176.233,10.006,148.980
C03289=1145.578,411.157,-89.010,-176.234,10.008,148.981
C03290=1145.574,411.404,-89.047,-176.234,10.010,148.982
C03291=1145.570,411.652,-89.085,-176.235,10.012,148.983
C03292=1145.566,411.899,-89.122,-176.236,10.014,148.983
C03293=1145.562,412.146,-89.159,-176.237,10.016,148.984
C03294=1145.559,412.394,-89.196,-176.238,10.017,148.985
C03295=1145.555,412.640,-89.233,-176.239,10.019,148.985
C03296=1145.552,412.887,-89.270,-176.240,10.021,148.986
C03297=1145.547,413.134,-89.307,-176.241,10.023,148.987
C03298=1145.544,413.382,-89.344,-176.241,10.026,148.988
C03299=1145.540,413.629,-89.381,-176.242,10.028,148.988
C03300=1145.536,413.876,-89.418,-176.243,10.030,148.989
C03301=1145.532,414.123,-89.455,-176.244,10.032,148.990
C03302=1145.528,414.371,-89.492,-176.244,10.033,148.991
C03303=1145.525,414.618,-89.530,-176.245,10.035,148.991
C03304=1145.521,414.866,-89.567,-176.245,10.038,148.992
C03305=1145.519,415.112,-89.604,-176.246,10.040,148.993
C03306=1145.517,415.360,-89.640,-176.247,10.042,148.993
C03307=1145.516,415.600,-89.677,-176.248,10.044,148.994
C03308=1145.516,415.841,-89.712,-176.248,10.045,148.995
C03309=1145.516,416.081,-89.748,-176.249,10.047,148.995
C03310=1145.517,416.322,-89.784,-176.249,10.050,148.996
C03311=1145.518,416.561,-89.818,-176.250,10.052,148.997
C03312=1145.521,416.802,-89.854,-176.251,10.053,148.997
C03313=1145.523,417.041,-89.889,-176.251,10.055,148.998
C03314=1145.527,417.280,-89.924,-176.252,10.057,148.999
C03315=1145.106,417.283,-89.974,-176.254,10.068,149.002
C03316=1145.103,417.041,-89.939,-176.254,10.066,149.002
C03317=1145.100,416.800,-89.903,-176.253,10.064,149.001
C03318=1145.098,416.558,-89.868,-176.252,10.062,149.000
C03319=1145.096,416.317,-89.832,-176.252,10.060,149.000
C03320=1145.095,416.075,-89.796,-176.251,10.059,148.999
C03321=1145.095,415.833,-89.760,-176.250,10.057,148.998
C03322=1145.095,415.590,-89.724,-176.249,10.055,148.998
C03323=1145.096,415.348,-89.688,-176.249,10.052,148.997
C03324=1145.098,415.101,-89.652,-176.249,10.051,148.996
C03325=1145.101,414.854,-89.614,-176.248,10.049,148.995
C03326=1145.104,414.606,-89.578,-176.247,10.047,148.995
C03327=1145.107,414.360,-89.540,-176.246,10.045,148.994
C03328=1145.112,414.112,-89.503,-176.246,10.042,148.993
C03329=1145.115,413.864,-89.466,-176.245,10.040,148.992
C03330=1145.119,413.617,-89.429,-176.244,10.038,148.992
C03331=1145.123,413.371,-89.392,-176.243,10.036,148.991
C03332=1145.127,413.123,-89.355,-176.242,10.034,148.990
C03333=1145.131,412.876,-89.318,-176.242,10.033,148.990
C03334=1145.135,412.628,-89.281,-176.240,10.031,148.989
C03335=1145.138,412.382,-89.243,-176.240,10.028,148.988
C03336=1145.142,412.134,-89.206,-176.239,10.026,148.987
C03337=1145.146,411.887,-89.169,-176.238,10.024,148.986
C03338=1145.150,411.640,-89.131,-176.238,10.022,148.986
C03339=1145.154,411.393,-89.095,-176.236,10.020,148.985
C03340=1145.157,411.145,-89.057,-176.236,10.018,148.984
C03341=1145.161,410.898,-89.020,-176.235,10.016,148.984
C03342=1145.165,410.652,-88.984,-176.234,10.015,148.983
C03343=1145.169,410.404,-88.947,-176.233,10.013,148.982
C03344=1145.172,410.157,-88.909,-176.232,10.010,148.981
C03345=1145.176,409.909,-88.873,-176.231,10.009,148.981
C03346=1145.180,409.663,-88.835,-176.230,10.007,148.980
C03347=1145.184,409.416,-88.798,-176.229,10.005,148.979
C03348=1145.188,409.168,-88.761,-176.228,10.003,148.978
C03349=1145.192,408.921,-88.724,-176.227,10.001,148.977
C03350=1145.195,408.674,-88.686,-176.227,9.999,148.977
C03351=1145.199,408.426,-88.649,-176.226,9.997,148.976
C03352=1145.203,408.179,-88.612,-176.224,9.995,148.975
C03353=1145.207,407.932,-88.576,-176.223,9.993,148.974
C03354=1145.211,407.685,-88.538,-176.223,9.991,148.974
C03355=1145.214,407.437,-88.501,-176.222,9.989,148.973
C03356=1145.218,407.190,-88.464,-176.221,9.987,148.972
C03357=1145.222,406.943,-88.428,-176.220,9.985,148.971
C03358=1145.226,406.697,-88.390,-176.219,9.983,148.971
C03359=1145.229,406.449,-88.353,-176.217,9.982,148.970
C03360=1145.233,406.202,-88.316,-176.216,9.980,148.969
C03361=1145.237,405.954,-88.279,-176.215,9.978,148.968
C03362=1145.241,405.707,-88.241,-176.214,9.976,148.967
C03363=1145.245,405.460,-88.204,-176.213,9.974,148.967
C03364=1145.249,405.213,-88.167,-176.212,9.972,148.966
C03365=1145.253,404.965,-88.131,-176.211,9.970,148.965
C03366=1145.256,404.718,-88.093,-176.210,9.968,148.964
C03367=1145.260,404.471,-88.056,-176.209,9.967,148.964
C03368=1145.264,404.224,-88.019,-176.207,9.965,148.963
C03369=1145.268,403.977,-87.983,-176.206,9.963,148.962
C03370=1145.271,403.729,-87.945,-176.205,9.961,148.961
C03371=1145.275,403.482,-87.908,-176.204,9.959,148.960
C03372=1145.279,403.235,-87.871,-176.203,9.956,148.959
C03373=1145.282,402.987,-87.834,-176.202,9.954,148.959
C03374=1145.287,402.740,-87.797,-176.200,9.953,148.958
C03375=1145.290,402.494,-87.759,-176.200,9.951,148.957
C03376=1145.294,402.246,-87.722,-176.199,9.949,148.956
C03377=1145.298,401.999,-87.685,-176.197,9.947,148.955
C03378=1145.302,401.751,-87.648,-176.196,9.945,148.955
C03379=1145.306,401.505,-87.611,-176.195,9.943,148.954
C03380=1145.310,401.258,-87.574,-176.194,9.941,148.953
C03381=1145.313,401.010,-87.537,-176.193,9.940,148.952
C03382=1145.317,400.763,-87.500,-176.191,9.938,148.951
C03383=1145.320,400.516,-87.463,-176.190,9.936,148.951
C03384=1145.324,400.268,-87.426,-176.189,9.934,148.950
C03385=1145.328,400.021,-87.389,-176.188,9.932,148.949
C03386=1145.332,399.774,-87.352,-176.187,9.930,148.948
C03387=1145.336,399.527,-87.314,-176.186,9.927,148.947
C03388=1145.339,399.280,-87.277,-176.185,9.925,148.946
C03389=1145.344,399.032,-87.240,-176.184,9.923,148.945
C03390=1145.348,398.785,-87.203,-176.183,9.921,148.945
C03391=1145.351,398.539,-87.166,-176.181,9.920,148.944
C03392=1145.355,398.291,-87.129,-176.180,9.918,148.943
C03393=1145.359,398.043,-87.092,-176.179,9.916,148.942
C03394=1145.363,397.796,-87.055,-176.178,9.914,148.941
C03395=1145.366,397.549,-87.017,-176.177,9.912,148.941
C03396=1145.370,397.302,-86.981,-176.175,9.910,148.940
C03397=1145.374,397.055,-86.944,-176.174,9.908,148.939
C03398=1145.378,396.808,-86.907,-176.173,9.906,148.938
C03399=1145.381,396.561,-86.869,-176.172,9.904,148.937
C03400=1145.385,396.313,-86.832,-176.171,9.902,148.936
C03401=1145.389,396.066,-86.795,-176.170,9.899,148.936
C03402=1145.393,395.819,-86.759,-176.169,9.897,148.935
C03403=1145.397,395.572,-86.721,-176.168,9.895,148.934
C03404=1145.401,395.324,-86.684,-176.167,9.892,148.933
C03405=1145.405,395.077,-86.647,-176.166,9.890,148.932
C03406=1145.409,394.830,-86.610,-176.165,9.888,148.931
C03407=1145.412,394.583,-86.572,-176.164,9.886,148.930
C03408=1145.416,394.336,-86.535,-176.163,9.883,148.930
C03409=1145.419,394.089,-86.499,-176.162,9.881,148.929
C03410=1145.423,393.841,-86.462,-176.161,9.879,148.928
C03411=1145.427,393.594,-86.425,-176.161,9.878,148.927
C03412=1145.431,393.347,-86.387,-176.160,9.875,148.926
C03413=1145.435,393.100,-86.350,-176.159,9.873,148.926
C03414=1145.438,392.852,-86.313,-176.158,9.871,148.925
C03415=1145.442,392.605,-86.276,-176.157,9.868,148.924
C03416=1145.446,392.358,-86.239,-176.156,9.866,148.923
C03417=1145.450,392.111,-86.202,-176.156,9.863,148.922
C03418=1145.454,391.863,-86.165,-176.155,9.861,148.921
C03419=1145.458,391.616,-86.128,-176.155,9.858,148.921
C03420=1145.462,391.330,-86.085,-176.154,9.855,148.919
C03421=1145.466,391.042,-86.042,-176.153,9.853,148.919
C03422=1145.471,390.755,-85.999,-176.152,9.850,148.918
C03423=1145.475,390.469,-85.956,-176.151,9.847,148.917
C03424=1145.479,390.221,-85.919,-176.151,9.844,148.916
C03425=1145.483,389.974,-85.882,-176.150,9.841,148.915
C03426=1145.487,389.727,-85.845,-176.150,9.838,148.914
C03427=1145.491,389.480,-85.807,-176.149,9.837,148.914
C03428=1145.494,389.232,-85.770,-176.149,9.834,148.913
C03429=1145.497,388.986,-85.734,-176.148,9.831,148.912
C03430=1145.502,388.738,-85.697,-176.148,9.828,148.911
C03431=1145.506,388.491,-85.660,-176.148,9.826,148.910
C03432=1145.509,388.244,-85.622,-176.148,9.822,148.909
C03433=1145.513,387.997,-85.585,-176.148,9.819,148.908
C03434=1145.517,387.749,-85.549,-176.147,9.817,148.908
C03435=1145.521,387.502,-85.512,-176.147,9.814,148.907
C03436=1145.524,387.255,-85.475,-176.147,9.811,148.906
C03437=1145.528,387.008,-85.438,-176.147,9.808,148.905
C03438=1145.532,386.761,-85.401,-176.147,9.805,148.905
C03439=1145.536,386.514,-85.364,-176.147,9.802,148.904
C03440=1145.539,386.266,-85.327,-176.147,9.799,148.903
C03441=1145.543,386.019,-85.290,-176.148,9.796,148.902
C03442=1145.548,385.771,-85.253,-176.148,9.793,148.902
C03443=1145.551,385.525,-85.217,-176.148,9.790,148.901
C03444=1145.555,385.277,-85.180,-176.149,9.786,148.900
C03445=1145.558,385.030,-85.143,-176.149,9.783,148.899
C03446=1145.562,384.783,-85.105,-176.150,9.780,148.899
C03447=1145.566,384.536,-85.068,-176.150,9.776,148.898
C03448=1145.570,384.289,-85.031,-176.151,9.773,148.897
C03449=1145.573,384.041,-84.995,-176.151,9.770,148.897
C03450=1145.577,383.794,-84.958,-176.152,9.766,148.896
C03451=1145.581,383.547,-84.921,-176.152,9.763,148.895
C03452=1145.585,383.299,-84.884,-176.154,9.759,148.894
C03453=1145.590,383.052,-84.847,-176.154,9.756,148.894
C03454=1145.592,382.805,-84.811,-176.155,9.753,148.893
C03455=1145.596,382.557,-84.774,-176.156,9.749,148.892
C03456=1145.601,382.310,-84.737,-176.157,9.746,148.892
C03457=1145.605,382.063,-84.700,-176.159,9.742,148.891
C03458=1145.608,381.816,-84.664,-176.160,9.737,148.890
C03459=1145.611,381.568,-84.627,-176.161,9.734,148.890
C03460=1145.616,381.321,-84.590,-176.162,9.730,148.889
C03461=1145.620,381.074,-84.553,-176.164,9.727,148.889
C03462=1145.623,380.827,-84.517,-176.165,9.723,148.888
C03463=1145.627,380.580,-84.480,-176.167,9.719,148.887
C03464=1145.631,380.333,-84.443,-176.168,9.715,148.887
C03465=1145.635,380.085,-84.406,-176.170,9.711,148.886
C03466=1145.638,379.837,-84.370,-176.171,9.707,148.885
C03467=1145.642,379.590,-84.333,-176.173,9.703,148.885
C03468=1145.647,379.343,-84.296,-176.174,9.699,148.884
C03469=1145.650,379.096,-84.260,-176.176,9.696,148.884
C03470=1145.654,378.849,-84.223,-176.178,9.691,148.883
C03471=1145.658,378.602,-84.186,-176.180,9.687,148.883
C03472=1145.661,378.355,-84.150,-176.181,9.683,148.882
C03473=1145.665,378.106,-84.114,-176.183,9.680,148.882
C03474=1145.669,377.859,-84.077,-176.185,9.675,148.881
C03475=1145.673,377.612,-84.040,-176.187,9.672,148.880
C03476=1145.677,377.365,-84.004,-176.189,9.667,148.880
C03477=1145.681,377.117,-83.967,-176.191,9.663,148.879
C03478=1145.685,376.870,-83.931,-176.193,9.659,148.879
C03479=1145.689,376.623,-83.894,-176.195,9.655,148.878
C03480=1145.692,376.376,-83.858,-176.198,9.651,148.878
C03481=1145.696,376.128,-83.822,-176.199,9.647,148.877
C03482=1145.700,375.881,-83.785,-176.202,9.642,148.877
C03483=1145.704,375.634,-83.749,-176.203,9.639,148.876
C03484=1145.708,375.386,-83.712,-176.206,9.634,148.876
C03485=1145.711,375.139,-83.676,-176.208,9.630,148.875
C03486=1145.715,374.892,-83.639,-176.210,9.626,148.875
C03487=1145.719,374.644,-83.604,-176.212,9.622,148.874
C03488=1145.723,374.397,-83.567,-176.215,9.617,148.874
C03489=1145.727,374.150,-83.531,-176.217,9.614,148.873
C03490=1145.731,373.902,-83.494,-176.219,9.609,148.873
C03491=1145.734,373.655,-83.458,-176.222,9.605,148.872
C03492=1145.738,373.408,-83.422,-176.224,9.601,148.872
C03493=1145.742,373.161,-83.386,-176.226,9.597,148.872
C03494=1145.746,372.913,-83.350,-176.229,9.593,148.871
C03495=1145.749,372.666,-83.313,-176.231,9.588,148.871
C03496=1145.754,372.418,-83.277,-176.234,9.584,148.870
C03497=1145.757,372.171,-83.241,-176.236,9.581,148.870
C03498=1145.762,371.924,-83.205,-176.239,9.576,148.869
C03499=1145.765,371.676,-83.169,-176.241,9.572,148.869
C03500=1145.769,371.429,-83.132,-176.244,9.567,148.868
C03501=1145.773,371.181,-83.097,-176.246,9.563,148.868
C03502=1145.776,370.935,-83.061,-176.249,9.559,148.868
C03503=1145.781,370.687,-83.024,-176.251,9.555,148.867
C03504=1145.784,370.439,-82.989,-176.253,9.551,148.867
C03505=1145.788,370.192,-82.953,-176.256,9.547,148.867
C03506=1145.792,369.945,-82.916,-176.259,9.542,148.866
C03507=1145.796,369.698,-82.881,-176.261,9.538,148.866
C03508=1145.801,369.451,-82.844,-176.264,9.534,148.865
C03509=1145.804,369.203,-82.809,-176.267,9.530,148.865
C03510=1145.808,368.956,-82.773,-176.269,9.525,148.864
C03511=1145.812,368.708,-82.737,-176.272,9.522,148.864
C03512=1145.816,368.461,-82.701,-176.274,9.518,148.864
C03513=1145.819,368.213,-82.665,-176.277,9.513,148.863
C03514=1145.823,367.966,-82.630,-176.280,9.509,148.863
C03515=1145.827,367.718,-82.594,-176.282,9.505,148.863
C03516=1145.831,367.471,-82.558,-176.285,9.501,148.862
C03517=1145.835,367.224,-82.522,-176.287,9.496,148.862
C03518=1145.839,366.977,-82.487,-176.290,9.492,148.862
C03519=1145.843,366.729,-82.451,-176.292,9.489,148.861
C03520=1145.847,366.482,-82.415,-176.295,9.484,148.861
C03521=1145.850,366.234,-82.379,-176.298,9.480,148.860
C03522=1145.854,365.987,-82.344,-176.300,9.476,148.860
C03523=1145.858,365.739,-82.308,-176.303,9.472,148.860
C03524=1145.863,365.455,-82.267,-176.306,9.466,148.859
C03525=1145.867,365.172,-82.226,-176.309,9.462,148.859
C03526=1145.872,364.889,-82.185,-176.312,9.457,148.858
C03527=1145.876,364.605,-82.145,-176.315,9.453,148.858
C03528=1145.880,364.358,-82.109,-176.318,9.449,148.858
C03529=1145.884,364.111,-82.074,-176.321,9.445,148.857
C03530=1145.888,363.863,-82.038,-176.323,9.440,148.857
C03531=1145.891,363.616,-82.003,-176.325,9.437,148.857
C03532=1145.895,363.368,-81.967,-176.328,9.433,148.856
C03533=1145.899,363.120,-81.932,-176.331,9.428,148.856
C03534=1145.904,362.873,-81.897,-176.333,9.424,148.856
C03535=1145.908,362.626,-81.861,-176.336,9.420,148.855
C03536=1145.911,362.378,-81.826,-176.338,9.416,148.855
C03537=1145.915,362.131,-81.790,-176.341,9.412,148.855
C03538=1145.919,361.884,-81.755,-176.344,9.408,148.854
C03539=1145.923,361.636,-81.719,-176.346,9.404,148.854
C03540=1145.927,361.388,-81.684,-176.349,9.400,148.854
C03541=1145.931,361.141,-81.649,-176.351,9.396,148.853
C03542=1145.935,360.894,-81.614,-176.354,9.392,148.853
C03543=1145.938,360.646,-81.578,-176.357,9.388,148.852
C03544=1145.942,360.398,-81.543,-176.360,9.384,148.852
C03545=1145.946,360.151,-81.508,-176.362,9.380,148.852
C03546=1145.950,359.904,-81.473,-176.364,9.376,148.852
C03547=1145.954,359.656,-81.438,-176.367,9.372,148.851
C03548=1145.958,359.408,-81.402,-176.369,9.368,148.851
C03549=1145.962,359.162,-81.367,-176.372,9.364,148.850
C03550=1145.966,358.914,-81.332,-176.375,9.360,148.850
C03551=1145.969,358.666,-81.297,-176.377,9.356,148.850
C03552=1145.973,358.419,-81.262,-176.380,9.352,148.849
C03553=1145.977,358.171,-81.227,-176.382,9.348,148.849
C03554=1145.981,357.924,-81.192,-176.385,9.344,148.849
C03555=1145.985,357.676,-81.157,-176.387,9.340,148.848
C03556=1145.989,357.429,-81.122,-176.390,9.336,148.848
C03557=1145.993,357.181,-81.087,-176.393,9.332,148.848
C03558=1145.998,356.934,-81.052,-176.395,9.328,148.847
C03559=1146.002,356.686,-81.017,-176.397,9.324,148.847
C03560=1146.004,356.439,-80.982,-176.399,9.321,148.847
C03561=1146.009,356.191,-80.947,-176.402,9.317,148.846
C03562=1146.013,355.944,-80.912,-176.405,9.312,148.846
C03563=1146.017,355.696,-80.877,-176.407,9.309,148.846
C03564=1146.021,355.449,-80.842,-176.410,9.305,148.845
C03565=1146.025,355.201,-80.807,-176.413,9.300,148.845
C03566=1146.029,354.954,-80.773,-176.414,9.297,148.845
C03567=1146.032,354.706,-80.738,-176.417,9.293,148.844
C03568=1146.036,354.458,-80.703,-176.420,9.288,148.844
C03569=1146.041,354.211,-80.668,-176.422,9.285,148.844
C03570=1146.044,353.963,-80.633,-176.425,9.281,148.843
C03571=1146.048,353.716,-80.599,-176.427,9.278,148.843
C03572=1146.052,353.468,-80.564,-176.430,9.273,148.843
C03573=1146.057,353.221,-80.529,-176.432,9.269,148.842
C03574=1146.060,352.973,-80.495,-176.435,9.266,148.842
C03575=1146.064,352.726,-80.460,-176.437,9.261,148.842
C03576=1146.068,352.478,-80.425,-176.440,9.257,148.841
C03577=1146.072,352.230,-80.390,-176.442,9.254,148.841
C03578=1146.076,351.983,-80.356,-176.445,9.250,148.841
C03579=1146.080,351.735,-80.321,-176.447,9.246,148.841
C03580=1146.084,351.488,-80.287,-176.450,9.242,148.840
C03581=1146.087,351.240,-80.252,-176.453,9.238,148.840
C03582=1146.092,350.993,-80.217,-176.455,9.235,148.840
C03583=1146.096,350.745,-80.182,-176.458,9.230,148.839
C03584=1146.100,350.498,-80.148,-176.460,9.226,148.839
C03585=1146.104,350.250,-80.114,-176.462,9.223,148.839
C03586=1146.108,350.003,-80.080,-176.465,9.218,148.838
C03587=1146.111,349.754,-80.045,-176.468,9.215,148.838
C03588=1146.116,349.507,-80.010,-176.470,9.211,148.838
C03589=1146.120,349.260,-79.977,-176.473,9.207,148.837
C03590=1146.124,349.012,-79.942,-176.475,9.203,148.837
C03591=1146.128,348.765,-79.908,-176.478,9.199,148.837
C03592=1146.132,348.517,-79.873,-176.480,9.196,148.836
C03593=1146.136,348.269,-79.839,-176.483,9.191,148.836
C03594=1146.139,348.021,-79.804,-176.485,9.188,148.836
C03595=1146.144,347.774,-79.770,-176.488,9.184,148.836
C03596=1146.147,347.526,-79.736,-176.490,9.180,148.835
C03597=1146.152,347.279,-79.701,-176.493,9.176,148.835
C03598=1146.156,347.032,-79.667,-176.496,9.172,148.835
C03599=1146.160,346.783,-79.632,-176.498,9.169,148.834
C03600=1146.163,346.536,-79.599,-176.500,9.165,148.834
C03601=1146.167,346.288,-79.564,-176.503,9.161,148.834
C03602=1146.171,346.041,-79.530,-176.505,9.157,148.833
C03603=1146.176,345.793,-79.496,-176.508,9.153,148.833
C03604=1146.179,345.545,-79.462,-176.511,9.150,148.833
C03605=1146.184,345.298,-79.427,-176.513,9.145,148.832
C03606=1146.188,345.051,-79.394,-176.515,9.142,148.832
C03607=1146.192,344.803,-79.359,-176.518,9.138,148.832
C03608=1146.196,344.555,-79.326,-176.521,9.133,148.832
C03609=1146.199,344.307,-79.291,-176.523,9.130,148.831
C03610=1146.204,344.060,-79.257,-176.526,9.126,148.831
C03611=1146.208,343.813,-79.223,-176.528,9.123,148.831
C03612=1146.212,343.564,-79.189,-176.531,9.118,148.830
C03613=1146.216,343.317,-79.155,-176.533,9.115,148.830
C03614=1146.219,343.070,-79.121,-176.536,9.111,148.830
C03615=1146.224,342.822,-79.087,-176.538,9.108,148.830
C03616=1146.228,342.574,-79.053,-176.541,9.103,148.829
C03617=1146.231,342.327,-79.019,-176.544,9.099,148.829
C03618=1146.236,342.079,-78.986,-176.546,9.096,148.829
C03619=1146.240,341.831,-78.951,-176.549,9.092,148.828
C03620=1146.244,341.583,-78.918,-176.551,9.088,148.828
C03621=1146.248,341.336,-78.884,-176.554,9.084,148.828
C03622=1146.252,341.089,-78.850,-176.556,9.081,148.828
C03623=1146.256,340.840,-78.816,-176.559,9.077,148.827
C03624=1146.260,340.593,-78.782,-176.561,9.073,148.827
C03625=1146.264,340.345,-78.749,-176.564,9.069,148.827
C03626=1146.268,340.097,-78.714,-176.566,9.066,148.827
C03627=1146.272,339.849,-78.681,-176.569,9.062,148.826
C03628=1146.276,339.569,-78.643,-176.572,9.058,148.826
C03629=1146.282,339.289,-78.605,-176.575,9.054,148.826
C03630=1146.286,339.009,-78.567,-176.577,9.049,148.825
C03631=1146.290,338.728,-78.528,-176.580,9.045,148.825
C03632=1146.295,338.480,-78.495,-176.583,9.041,148.825
C03633=1146.298,338.233,-78.461,-176.586,9.037,148.825
C03634=1146.302,337.985,-78.428,-176.588,9.034,148.824
C03635=1146.307,337.737,-78.393,-176.591,9.029,148.824
C03636=1146.311,337.490,-78.360,-176.593,9.026,148.824
C03637=1146.315,337.242,-78.327,-176.596,9.022,148.823
C03638=1146.319,336.995,-78.293,-176.598,9.019,148.823
C03639=1146.322,336.746,-78.260,-176.601,9.015,148.823
C03640=1146.326,336.499,-78.226,-176.603,9.011,148.823
C03641=1146.330,336.251,-78.193,-176.606,9.007,148.822
C03642=1146.334,336.004,-78.159,-176.608,9.004,148.822
C03643=1146.339,335.756,-78.126,-176.611,8.999,148.822
C03644=1146.343,335.508,-78.092,-176.613,8.996,148.822
C03645=1146.347,335.260,-78.059,-176.616,8.992,148.822
C03646=1146.351,335.012,-78.025,-176.618,8.989,148.821
C03647=1146.355,334.765,-77.992,-176.621,8.984,148.821
C03648=1146.359,334.517,-77.959,-176.623,8.981,148.821
C03649=1146.363,334.269,-77.926,-176.626,8.977,148.820
C03650=1146.367,334.021,-77.892,-176.629,8.974,148.820
C03651=1146.371,333.774,-77.859,-176.632,8.970,148.820
C03652=1146.375,333.525,-77.826,-176.634,8.966,148.820
C03653=1146.379,333.278,-77.792,-176.636,8.962,148.819
C03654=1146.383,333.030,-77.759,-176.639,8.959,148.819
C03655=1146.387,332.783,-77.726,-176.642,8.955,148.819
C03656=1146.391,332.535,-77.692,-176.644,8.951,148.819
C03657=1146.395,332.287,-77.659,-176.647,8.947,148.818
C03658=1146.399,332.040,-77.626,-176.649,8.944,148.818
C03659=1146.404,331.792,-77.593,-176.652,8.940,148.818
C03660=1146.408,331.544,-77.560,-176.654,8.936,148.818
C03661=1146.412,331.296,-77.527,-176.656,8.933,148.817
